# B&R Automation Studio project NAELD004C00R10L518F00 (part 8)

#### Act_OptP0201QueryWorkOrderInfo.st
```iecst
ACTION Act_OptP0201QueryWorkOrderInfo:

	//Mask Magazine Barcode / SlotId
	IF p_tyNtParamCurr.bHermesSvyMagTypeMc = FALSE THEN
		fUIInRtStatOff(ADR(tyP0201OpsTravLifter.tyQueryWorkOrderInfo.tyBitmapMask.uiMaskRtStat)); //show the mask
	ELSE
		fUIInRtStatHide(ADR(tyP0201OpsTravLifter.tyQueryWorkOrderInfo.tyBitmapMask.uiMaskRtStat)); //hide the mask
	END_IF

	//Mask Barcode Scanner
	IF p_tyNtParamCurr.bHermesScannerPrep = TRUE AND p_tyMcParamCurr.bHermesScannerEn = TRUE THEN
		fUIInRtStatHide(ADR(tyP0201OpsTravLifter.tyQueryWorkOrderInfo.tyBtnBarcodeScanner.uiMaskRtStat)); //hide the mask
	ELSE
		fUIInRtStatOff(ADR(tyP0201OpsTravLifter.tyQueryWorkOrderInfo.tyBtnBarcodeScanner.uiMaskRtStat)); //show the mask
	END_IF

	IF 	EDGEPOS (tyP0201OpsTravLifter.tyQueryWorkOrderInfo.tyBtnBarcodeScanner.bValue = TRUE) THEN
		fUIInRtStatHide(ADR(tyP0201OpsTravLifter.tyQueryWorkOrderInfo.tyLyr.uiRtStat)); //hide popup QueryBoardInfo
		fUIInRtStatOff(ADR(tyP0201OpsTravLifter.tyBarcodeScanner.tyLyr.uiRtStat)); //show popup BCScanner
		fUIInRtStatHide(ADR(tyP0201OpsTravLifter.tyBarcodeScanner.tyBtnMagazine.uiMaskRtStat)); //hide Mask Magazine
		fUIInRtStatOff(ADR(tyP0201OpsTravLifter.tyBarcodeScanner.tyBtnTop.uiMaskRtStat)); //Mask Top
	END_IF

	//Convert
	iSlotId := DINT_TO_INT(tyP0201OpsTravLifter.tyQueryWorkOrderInfo.tyNumSlotId.diValue);

	//Press OK, set bQueryWorkOrderInfo
	IF	tyP0201OpsTravLifter.tyQueryWorkOrderInfo.tyBtnOk.bRtCompl = TRUE THEN

		fUIInRtStatHide(ADR(tyP0201OpsTravLifter.tyQueryWorkOrderInfo.tyLyr.uiRtStat)); //close popup

		IF (tyP0201OpsTravLifter.tyQueryWorkOrderInfo.tyStringMagazineId.sValue <> '') OR (iSlotId <> 0)
			OR (tyP0201OpsTravLifter.tyQueryWorkOrderInfo.tyStringBarcode.sValue <> '') THEN
			bQueryWorkOrderInfo := TRUE;
			tyP0201OpsTravLifter.tyCurrWorkOrderInfo.tyBtnQueryWorkOrderInfo.bValue := TRUE;
		ELSE
			bQueryWorkOrderInfo := FALSE;
			tyP0201OpsTravLifter.tyCurrWorkOrderInfo.tyBtnQueryWorkOrderInfo.bValue := FALSE;
		END_IF

		tyP0201OpsTravLifter.tyQueryWorkOrderInfo.tyBtnOk.bValue := FALSE;

		tyP0201OpsTravLifter.tyQueryWorkOrderInfo.tyBtnOk.bRtCompl := FALSE;

	END_IF

	//Press Cancel
	IF	tyP0201OpsTravLifter.tyQueryWorkOrderInfo.tyBtnCancel.bRtCompl = TRUE THEN

		fUIInRtStatHide(ADR(tyP0201OpsTravLifter.tyQueryWorkOrderInfo.tyLyr.uiRtStat)); //hide
		fUIInRtStatOff(ADR(tyP0201OpsTravLifter.tyCurrWorkOrderInfo.tyLyr.uiRtStat)); //hide

		tyP0201OpsTravLifter.tyQueryWorkOrderInfo.tyBtnCancel.bRtCompl := FALSE;
		tyP0201OpsTravLifter.tyQueryWorkOrderInfo.tyBtnCancel.bValue := FALSE;
	END_IF

END_ACTION
```

#### Act_OptP0201UpdtDat.st
```iecst
ACTION Act_OptP0201UpdtDat:

	//Status
	fbMcStatUpdtTm(IN := TRUE);
	IF fbMcStatUpdtTm.Q = TRUE THEN
		fbMcStatUpdtTm(IN := FALSE);

		IF p_bOpsTravLifLDAWPosDiff THEN
			IF p_tyNtParamCurr.bDSWidthChkPrep AND p_tyMcParamCurr.bDSWidthChkEn AND p_tyDI.bDSWidthChkSen=FALSE THEN
				tyP0201OpsTravLifter.tyOps.tyStringMcStat.sValue	:= 'Width Check Sensor Block Downstream';
			ELSIF p_tyNtParamCurr.bLFPrep AND p_tyMcParamCurr.bLFEn AND p_bLFFollowerDSAllow=FALSE THEN
				IF p_tyMcParamCurr.bSectionLeader THEN
					tyP0201OpsTravLifter.tyOps.tyStringMcStat.sValue	:= 'Section Leader: Block Downstream';
				ELSE
					tyP0201OpsTravLifter.tyOps.tyStringMcStat.sValue	:= 'Leader Issue Block Downstream';
				END_IF

			ELSE
				tyP0201OpsTravLifter.tyOps.tyStringMcStat.sValue	:= p_sOpsTravLifLDStepTxt;
			END_IF
		ELSE
			tyP0201OpsTravLifter.tyOps.tyStringMcStat.sValue	:= p_sOpsTravLifLDStepTxt;
		END_IF
	END_IF

	//Mode
	tyP0201OpsTravLifter.tyOps.tyTxtMod.usiValueIdx	:= p_tyProdRcpCurrRcp2.usiMcMod;

	//Width
	IF p_tyNtParamCurr.bAWPrep = TRUE AND p_tyMcParamCurr.bAWDis = FALSE THEN
		tyP0201OpsTravLifter.tyOps.tyNumWidth.diValue	:= p_tyMcParamCurr.diWidthAtHmPosInUM - p_diAWOpenActualPos;
		tyP0201OpsTravLifter.tyOps.tyNumWidth2.diValue	:= p_tyMcParamCurr.diWidthAtHmPosInUM - p_diAWOpenActualPos;
	ELSE
		tyP0201OpsTravLifter.tyOps.tyNumWidth.diValue	:= p_tyProdRcpCurrRcp2.diWidthInUM;
		tyP0201OpsTravLifter.tyOps.tyNumWidth2.diValue	:= p_tyProdRcpCurrRcp2.diWidthInUM2;
	END_IF

	//Product Info
	IF p_tyNtParamCurr.eProjMag <> LDMagQuadruple THEN
		IF p_tyNtParamCurr.bProjAutoRcpPrep AND p_tyMcParamCurr.bHermesSvyEn THEN
			IF p_ausiSvyMagAccOrder[1] = 10 THEN
				tyP0201OpsTravLifter.tyOps.tyNumMinSltRange.diValue		:= p_diLinkAutoRcpMag1MinSlt;
				tyP0201OpsTravLifter.tyOps.tyNumMaxSltRange.diValue		:= p_diLinkAutoRcpMag1MaxSlt;
				tyP0201OpsTravLifter.tyOps.tyNumPitch.diValue			:= p_diLinkAutoRcpMag1Pitch;
				tyP0201OpsTravLifter.tyOps.tyStringProdNm.sValue		:= p_tyAutoRcpMagRcp[1].sWorkOrderId;
			ELSIF p_ausiSvyMagAccOrder[2] = 10 THEN
				tyP0201OpsTravLifter.tyOps.tyNumMinSltRange.diValue		:= p_diLinkAutoRcpMag2MinSlt;
				tyP0201OpsTravLifter.tyOps.tyNumMaxSltRange.diValue		:= p_diLinkAutoRcpMag2MaxSlt;
				tyP0201OpsTravLifter.tyOps.tyNumPitch.diValue			:= p_diLinkAutoRcpMag2Pitch;
				tyP0201OpsTravLifter.tyOps.tyStringProdNm.sValue		:= p_tyAutoRcpMagRcp[2].sWorkOrderId;
			ELSIF p_ausiSvyMagAccOrder[3] = 10 THEN
				tyP0201OpsTravLifter.tyOps.tyNumMinSltRange.diValue		:= p_diLinkAutoRcpMag3MinSlt;
				tyP0201OpsTravLifter.tyOps.tyNumMaxSltRange.diValue		:= p_diLinkAutoRcpMag3MaxSlt;
				tyP0201OpsTravLifter.tyOps.tyNumPitch.diValue			:= p_diLinkAutoRcpMag3Pitch;
				tyP0201OpsTravLifter.tyOps.tyStringProdNm.sValue		:= p_tyAutoRcpMagRcp[3].sWorkOrderId;
			END_IF
		ELSE //standard
			tyP0201OpsTravLifter.tyOps.tyNumMinSltRange.diValue		:= p_tyProdRcpCurrRcp2.diMinSltValue;
			tyP0201OpsTravLifter.tyOps.tyNumMaxSltRange.diValue		:= p_tyProdRcpCurrRcp2.diMaxSltValue;
			tyP0201OpsTravLifter.tyOps.tyNumPitch.diValue			:= p_tyProdRcpCurrRcp2.diPitch;
			tyP0201OpsTravLifter.tyOps.tyStringProdNm.sValue		:= p_tyProdRcpCurrRcp2.sRcpNm;
		END_IF

		tyP0201OpsTravLifter.tyOps.tyBtnToptoBtm.bValue			:= p_tyProdRcpCurrRcp2.bTopToBtm;

		tyP0201OpsTravLifter.tyOps.tyNumPshrOffset.diValue		:= p_tyProdRcpCurrRcp2.diPshrOffset;
		tyP0201OpsTravLifter.tyOps.tyNumMtrPshrExtSpd.diValue	:= p_tyProdRcpCurrRcp2.diMtrPshrExtSpd;
		tyP0201OpsTravLifter.tyOps.tyNumMtrPshrExtTorq.diValue	:= p_tyProdRcpCurrRcp2.diMtrPshrExtTorq;

	ELSE //quadral
		tyP0201OpsTravLifter.tyOps.tyStringProdNm.sValue		:= p_tyProdRcpCurrRcp2.sRcpNm;
		tyP0201OpsTravLifter.tyOps.tyNumMinSltRange.diValue		:= p_tyProdRcpCurrRcp2.diMinSltValue;
		tyP0201OpsTravLifter.tyOps.tyNumMaxSltRange.diValue		:= p_tyProdRcpCurrRcp2.diMaxSltValue;
		tyP0201OpsTravLifter.tyOps.tyBtnToptoBtm.bValue			:= p_tyProdRcpCurrRcp2.bTopToBtm;
		tyP0201OpsTravLifter.tyOps.tyNumPitch.diValue			:= p_tyProdRcpCurrRcp2.diPitch;

		tyP0201OpsTravLifter.tyOps.tyNumMinSltRange.diValue		:= p_tyProdRcpCurrRcp2.diMinSltValue;
		tyP0201OpsTravLifter.tyOps.tyNumMaxSltRange.diValue		:= p_tyProdRcpCurrRcp2.diMaxSltValue;
		tyP0201OpsTravLifter.tyOps.tyNumPitch.diValue			:= p_tyProdRcpCurrRcp2.diPitch;
	END_IF

	//PCB Status
	IF p_bPullConvHvBrd = TRUE THEN
		tyP0201OpsTravLifter.tyOps.tyBitmapPCB.usiValueIdx	:= 1;
	ELSE
		tyP0201OpsTravLifter.tyOps.tyBitmapPCB.usiValueIdx	:= 0;
	END_IF

	//Product Recipe 254
	tyP0201OpsTravLifter.tyOps.tyHotspotShowLRcp.uiRtStat.0 := NOT(tyP0201OpsTravLifter.tyOps.tyStringProdNm.sValue <> '');

	IF tyP0201OpsTravLifter.tyOps.tyHotspotShowLRcp.bRtCompl = TRUE THEN
		tyP0201OpsTravLifter.tyOps.tyHotspotShowLRcp.bRtCompl := FALSE;

		fUIInRtStatOff(ADR(tyP0201OpsTravLifter.tyRcpPopUp.tyLyr.uiRtStat));

		tyP0201OpsTravLifter.tyRcpPopUp.tyStringInfo.sValue  := p_tyProdRcpCurrRcp1.sRcpNm;

	ELSIF tyP0201OpsTravLifter.tyRcpPopUp.tyHotspotClose.bRtCompl = TRUE THEN
		tyP0201OpsTravLifter.tyRcpPopUp.tyHotspotClose.bRtCompl := FALSE;

		fUIInRtStatHide(ADR(tyP0201OpsTravLifter.tyRcpPopUp.tyLyr.uiRtStat));

	END_IF

END_ACTION
```

#### Act_EntP0202Disp.st
```iecst
ACTION Act_EntP0202Disp:

	//Access Address
	p_tyC0004Navi ACCESS ADR(tyP0202OpsMag1.tyNaviBack);

	p_tyC0005Main ACCESS ADR(tyCommon.tyMain);

	p_tyC0007Notif ACCESS ADR(tyCommon.tyNotif);

	p_tyC0008MsgBox ACCESS ADR(tyP0202OpsMag1.tyMsgBoxHide);

	p_tyC0009Info ACCESS ADR(tyCommon.tyInfo);

	p_tyC0011RcpPopUp ACCESS ADR(tyP0202OpsMag1.tyRcpPopUp);

	p_tyP0202Ops ACCESS ADR(tyP0202OpsMag1.tyOps);
	p_tyP0202IOMonitor ACCESS ADR(tyP0202OpsMag1.tyIOMonitor);
	p_tyP0202BypsInitConv ACCESS ADR(tyP0202OpsMag1.tyBypsInitConv);
	p_tyP0202Param ACCESS ADR(tyP0202OpsMag1.tyParam);

	//Display
	fUIInRtStatHide(ADR(tyP0202OpsMag1.tyIOMonitor.tyLyr.uiRtStat));
	fUIInRtStatHide(ADR(tyP0202OpsMag1.tyParam.tyLyr.uiRtStat));

	tyP0202OpsMag1.tyOps.tyBtnChgParam.uiRtStat.0	:= NOT(p_tyMcParamCurr.bChgParamEn);
	tyP0202OpsMag1.tyParam.tyNumMaxSlt.diValueMax	:= p_tyMagRcpCurrRcp.diTtlSlt;

	IF p_tyNtParamCurr.bMagAutoVerifyPrep = FALSE THEN
		tyP0202OpsMag1.tyIOMonitor.tyBtnMag1FixedClmpRS.usiTxtIdx	:= 75;
		tyP0202OpsMag1.tyIOMonitor.tyBtnMag1FixedUnclmpRS.usiTxtIdx:= 75;
		tyP0202OpsMag1.tyIOMonitor.tyBtnMag1RmtClmpRS.usiTxtIdx	:= 0;
		tyP0202OpsMag1.tyIOMonitor.tyBtnMag1RmtUnclmpRS.usiTxtIdx:= 0;
		tyP0202OpsMag1.tyIOMonitor.tyBtnMag1FixedClampCtrl.usiTxtIdx:= 41;
		tyP0202OpsMag1.tyIOMonitor.tyBtnMag1RemoteClampCtrl.usiTxtIdx:= 18;
	ELSE
		tyP0202OpsMag1.tyIOMonitor.tyBtnMag1FixedClmpRS.usiTxtIdx	:= 75;
		tyP0202OpsMag1.tyIOMonitor.tyBtnMag1FixedUnclmpRS.usiTxtIdx:= 75;
		tyP0202OpsMag1.tyIOMonitor.tyBtnMag1RmtClmpRS.usiTxtIdx	:= 0;
		tyP0202OpsMag1.tyIOMonitor.tyBtnMag1RmtUnclmpRS.usiTxtIdx:= 0;
		tyP0202OpsMag1.tyIOMonitor.tyBtnMag1FixedClampCtrl.usiTxtIdx:= 41;
		tyP0202OpsMag1.tyIOMonitor.tyBtnMag1RemoteClampCtrl.usiTxtIdx:= 18;

	END_IF

	fUIInRtStatHide(ADR(tyP0202OpsMag1.tyOps.tyBtnAIVWifi.uiRtStat));
	fUIInRtStatHide(ADR(tyP0202OpsMag1.tyOps.tyTxtLblAIV.uiRtStat));

	tyP0202OpsMag1.tyParam.tyNumMaxSlt.diValueMax	:= p_tyMagRcpCurrRcp.diTtlSlt;

END_ACTION
```

#### Act_OptP0202UpdtDat.st
```iecst
ACTION Act_OptP0202UpdtDat:

	//Status
	fbMcStatUpdtTm(IN := TRUE);
	IF fbMcStatUpdtTm.Q = TRUE THEN
		fbMcStatUpdtTm(IN := FALSE);

		IF p_tyNtParamCurr.bProjLifterMagPlatform THEN
			tyP0202OpsMag1.tyOps.tyStringMcStat.sValue	:= p_sOpsLifMagLDStepTxt;
		ELSE
			tyP0202OpsMag1.tyOps.tyStringMcStat.sValue	:= p_sOpsMagConvLD1StepTxt;
		END_IF

	END_IF

	//Mode
	tyP0202OpsMag1.tyOps.tyTxtMod.usiValueIdx	:= p_tyProdRcpCurrRcp1.usiMcMod;

	//Width
	IF p_tyNtParamCurr.bAWPrep = TRUE AND p_tyMcParamCurr.bAWDis = FALSE THEN
		tyP0202OpsMag1.tyOps.tyNumWidth.diValue	:= p_tyMcParamCurr.diWidthAtHmPosInUM - p_diAWOpenActualPos;
		tyP0202OpsMag1.tyOps.tyNumWidth2.diValue	:= p_tyMcParamCurr.diWidthAtHmPosInUM - p_diAWOpenActualPos;
	ELSE
		tyP0202OpsMag1.tyOps.tyNumWidth.diValue	:= p_tyProdRcpCurrRcp1.diWidthInUM;
		tyP0202OpsMag1.tyOps.tyNumWidth2.diValue	:= p_tyProdRcpCurrRcp1.diWidthInUM2;
	END_IF

	//Program Info
	IF p_tyNtParamCurr.eProjMag <> LDMagQuadruple THEN
		IF p_tyNtParamCurr.bProjAutoRcpPrep AND p_tyMcParamCurr.bHermesSvyEn THEN
			tyP0202OpsMag1.tyOps.tyNumMinSltRange.diValue		:= p_diLinkAutoRcpMag1MinSlt;
			tyP0202OpsMag1.tyOps.tyNumMaxSltRange.diValue		:= p_diLinkAutoRcpMag1MaxSlt;
			tyP0202OpsMag1.tyOps.tyNumPitch.diValue				:= p_diLinkAutoRcpMag1Pitch;
			tyP0202OpsMag1.tyOps.tyStringProdNm.sValue			:= p_tyAutoRcpMagRcp[1].sWorkOrderId;
		ELSE
			tyP0202OpsMag1.tyOps.tyNumMinSltRange.diValue		:= p_tyProdRcpCurrRcp2.diMinSltValue;
			tyP0202OpsMag1.tyOps.tyNumMaxSltRange.diValue		:= p_tyProdRcpCurrRcp2.diMaxSltValue;
			tyP0202OpsMag1.tyOps.tyNumPitch.diValue				:= p_tyProdRcpCurrRcp2.diPitch;
			tyP0202OpsMag1.tyOps.tyStringProdNm.sValue		:= p_tyProdRcpCurrRcp2.sRcpNm;
		END_IF
		tyP0202OpsMag1.tyOps.tyBtnToptoBtm.bValue			:= p_tyProdRcpCurrRcp2.bTopToBtm;
		//Magazine Info
		tyP0202OpsMag1.tyOps.tyStringMagNm.sValue	:= p_tyMagRcpCurrRcp.sRcpNm;
	ELSE
		CASE p_tyProdRcpCurrRcp2.usiMcMod OF
			0,2:
				tyP0202OpsMag1.tyOps.tyStringProdNm.sValue		:= p_tyProdRcpCurrRcp2.sRcpNm;
				tyP0202OpsMag1.tyOps.tyNumMinSltRange.diValue		:= p_tyProdRcpCurrRcp2.diMinSltValue;
				tyP0202OpsMag1.tyOps.tyNumMaxSltRange.diValue		:= p_tyProdRcpCurrRcp2.diMaxSltValue;
				tyP0202OpsMag1.tyOps.tyBtnToptoBtm.bValue			:= p_tyProdRcpCurrRcp2.bTopToBtm;
				tyP0202OpsMag1.tyOps.tyNumPitch.diValue			:= p_tyProdRcpCurrRcp2.diPitch;
				//Magazine Info
				tyP0202OpsMag1.tyOps.tyStringMagNm.sValue	:= p_tyMagRcpCurrRcp.sRcpNm;
			1:

				tyP0202OpsMag1.tyOps.tyStringProdNm.sValue		:= p_tyProdRcpCurrRcp2.sRcpNm;
				tyP0202OpsMag1.tyOps.tyNumMinSltRange.diValue		:= p_tyProdRcpCurrRcp2.diMinSltValueRear;
				tyP0202OpsMag1.tyOps.tyNumMaxSltRange.diValue		:= p_tyProdRcpCurrRcp2.diMaxSltValueRear;
				tyP0202OpsMag1.tyOps.tyBtnToptoBtm.bValue			:= p_tyProdRcpCurrRcp2.bTopToBtm;
				tyP0202OpsMag1.tyOps.tyNumPitch.diValue			:= p_tyProdRcpCurrRcp2.diPitchRear;
				//Magazine Info
				tyP0202OpsMag1.tyOps.tyStringMagNm.sValue	:= p_tyMagRcpCurrRcp1.sRcpNm;
		END_CASE
	END_IF
	//Magazine Info
//	tyP0202OpsMag1.tyOps.tyStringMagNm.sValue	:= p_tyMagRcpCurrRcp.sRcpNm;

	IF p_bBuffer1MagPresent = TRUE THEN
		tyP0202OpsMag1.tyOps.tyNumMag1AvlQty.diValue	:= p_tyBuffer1BffrStat.diTtlGdBrd + p_tyBuffer1BffrStat.diTtlBadBrd;
		tyP0202OpsMag1.tyOps.tyNumMag1TtlSlt.diValue	:= p_tyBuffer1BffrStat.diTtlBrdCap;
	ELSE
		tyP0202OpsMag1.tyOps.tyNumMag1AvlQty.diValue	:= 0;
		tyP0202OpsMag1.tyOps.tyNumMag1TtlSlt.diValue	:= 0;
	END_IF

	//Magazine Present States
	IF p_bBuffer1MagPresent = TRUE THEN

		IF p_tyBuffer1BffrStat.bBffrFull = TRUE THEN
			tyP0202OpsMag1.tyOps.tyTxtMag1Stat.usiValueIdx := 2;
			tyP0202OpsMag1.tyOps.tyTxtMag1Stat.usiColor	   := 0;
		ELSIF p_tyBuffer1BffrStat.bBffrMty = TRUE THEN
			tyP0202OpsMag1.tyOps.tyTxtMag1Stat.usiValueIdx := 1;
			tyP0202OpsMag1.tyOps.tyTxtMag1Stat.usiColor	   := 1;
		ELSE
			tyP0202OpsMag1.tyOps.tyTxtMag1Stat.usiValueIdx := 3;
			tyP0202OpsMag1.tyOps.tyTxtMag1Stat.usiColor	   := 0;
		END_IF

	ELSE
		tyP0202OpsMag1.tyOps.tyTxtMag1Stat.usiValueIdx := 0;
		tyP0202OpsMag1.tyOps.tyTxtMag1Stat.usiColor	   := 1;
	END_IF

	//Product Recipe 254
	tyP0202OpsMag1.tyOps.tyHotspotShowLRcp.uiRtStat.0 := NOT(tyP0202OpsMag1.tyOps.tyStringProdNm.sValue <> '');

	IF tyP0202OpsMag1.tyOps.tyHotspotShowLRcp.bRtCompl = TRUE THEN
		tyP0202OpsMag1.tyOps.tyHotspotShowLRcp.bRtCompl := FALSE;

		fUIInRtStatOff(ADR(tyP0202OpsMag1.tyRcpPopUp.tyLyr.uiRtStat));

		tyP0202OpsMag1.tyRcpPopUp.tyStringInfo.sValue  := p_tyProdRcpCurrRcp1.sRcpNm;

	ELSIF tyP0202OpsMag1.tyRcpPopUp.tyHotspotClose.bRtCompl = TRUE THEN
		tyP0202OpsMag1.tyRcpPopUp.tyHotspotClose.bRtCompl := FALSE;

		fUIInRtStatHide(ADR(tyP0202OpsMag1.tyRcpPopUp.tyLyr.uiRtStat));

	END_IF

END_ACTION
```

#### Act_OptP0202IOMonitor.st
```iecst
ACTION Act_OptP0202IOMonitor:

	IF tyP0202OpsMag1.tyOps.tyHotspotIOMonitor.bRtCompl = TRUE THEN
		tyP0202OpsMag1.tyOps.tyHotspotIOMonitor.bRtCompl	:= FALSE;

		fUIInRtStatOff(ADR(tyP0202OpsMag1.tyIOMonitor.tyLyr.uiRtStat));

		p_tyC0004Navi ACCESS ADR(tyP0202OpsMag1.tyNaviHide);

	ELSIF tyP0202OpsMag1.tyIOMonitor.tyHotspotClose.bRtCompl = TRUE THEN
		tyP0202OpsMag1.tyIOMonitor.tyHotspotClose.bRtCompl	:= FALSE;

		fUIInRtStatHide(ADR(tyP0202OpsMag1.tyIOMonitor.tyLyr.uiRtStat));

		p_tyC0004Navi ACCESS ADR(tyP0202OpsMag1.tyNaviBack);

	END_IF

	IF tyP0202OpsMag1.tyIOMonitor.tyLyr.uiRtStat.0 = FALSE THEN

		//Digital Input
		tyP0202OpsMag1.tyIOMonitor.tyBtnSafetyRlySig.bValue				:= p_tyDI.bSafetyRlySig;
		tyP0202OpsMag1.tyIOMonitor.tyBtnEStop.bValue					:= p_tyDI.bEStopSig;
		tyP0202OpsMag1.tyIOMonitor.tyBtnCoverSWSig.bValue				:= p_tyDI.bCoverSWSig;
		tyP0202OpsMag1.tyIOMonitor.tyBtnDSBA.bValue						:= p_tyDI.bDSBA;
		tyP0202OpsMag1.tyIOMonitor.tyBtnDSBB.bValue						:= p_tyDI.bDSBB;
		tyP0202OpsMag1.tyIOMonitor.tyBtnMag1FixedClmpRS.bValue			:= p_tyDI.bMag1FixedClampRS;
		tyP0202OpsMag1.tyIOMonitor.tyBtnMag1FixedUnclmpRS.bValue		:= p_tyDI.bMag1FixedUnclampRS;
		tyP0202OpsMag1.tyIOMonitor.tyBtnMag1RmtClmpRS.bValue			:= p_tyDI.bMag1RemoteClampRS;
		tyP0202OpsMag1.tyIOMonitor.tyBtnMag1RmtUnclmpRS.bValue			:= p_tyDI.bMag1RemoteUnclampRS;
		tyP0202OpsMag1.tyIOMonitor.tyBtnMag1ConvEntrySen.bValue			:= p_tyDI.bMagConvEntSen1;
		tyP0202OpsMag1.tyIOMonitor.tyBtnMag1PresentSen.bValue			:= p_tyDI.bMagPresentSen1;
		tyP0202OpsMag1.tyIOMonitor.tyBtnMag1AIVInPosSen1.bValue			:= p_tyDI.bMag1AGVInPosSen1;
		tyP0202OpsMag1.tyIOMonitor.tyBtnMag1AIVInPosSen2.bValue			:= p_tyDI.bMag1AGVInPosSen2;
		tyP0202OpsMag1.tyIOMonitor.tyBtnMag1OrientationChkSen1.bValue	:= p_tyDI.bMag1OrientChkSen1;
		tyP0202OpsMag1.tyIOMonitor.tyBtnMag1OrientationChkSen2.bValue	:= p_tyDI.bMag1OrientChkSen2;

		tyP0202OpsMag1.tyIOMonitor.tyBtnSelUnclampRS.bValue				:= p_tyDI.bMag1SelUnClampRS;

		tyP0202OpsMag1.tyIOMonitor.tyBtnCAB717Sen.bValue				:= p_tyDI.bMagConvCAB717MagSen1;
		tyP0202OpsMag1.tyIOMonitor.tyBtnHeightSen.bValue				:= p_tyDI.bMagConvHeightSen1 OR p_tyDI.bHighMagDetSen1;
		tyP0202OpsMag1.tyIOMonitor.tyBtnMagSmallSen.bValue				:= p_tyDI.bMagConvSmallMagSen1;
		tyP0202OpsMag1.tyIOMonitor.tyBtnMagLargeSen.bValue				:= p_tyDI.bMagConvLargeMagSen1;
		tyP0202OpsMag1.tyIOMonitor.tyBtnMagDetSen.bValue				:= p_tyDI.bMag1FixedSideDetect;
		tyP0202OpsMag1.tyIOMonitor.tyBtnTrllyExtRS.bValue				:= p_tyDI.bTrolleyExtRS1;
		tyP0202OpsMag1.tyIOMonitor.tyBtnTrllyPresentSen.bValue			:= p_tyDI.bTrolleyPreSen1;
		tyP0202OpsMag1.tyIOMonitor.tyBtnSltLckSen.bValue				:= p_tyDI.bSlotLckSenMag1;

		//Digital Output
		tyP0202OpsMag1.tyIOMonitor.tyBtnSafetyRlyRst.bValue				:= p_tyDO.bSafetyRlyRst;
		tyP0202OpsMag1.tyIOMonitor.tyBtnTLGreen.bValue					:= p_tyDO.bTLGreen;
		tyP0202OpsMag1.tyIOMonitor.tyBtnTLAmber.bValue					:= p_tyDO.bTLAmber;
		tyP0202OpsMag1.tyIOMonitor.tyBtnTLRed.bValue					:= p_tyDO.bTLRed;
		tyP0202OpsMag1.tyIOMonitor.tyBtnBuzzer.bValue					:= p_tyDO.bBuzzer;
		tyP0202OpsMag1.tyIOMonitor.tyBtnDBAA.bValue						:= p_tyDO.bDBAA;
		tyP0202OpsMag1.tyIOMonitor.tyBtnDBAB.bValue						:= p_tyDO.bDBAB;
		tyP0202OpsMag1.tyIOMonitor.tyBtnMag1FixedClampCtrl.bValue		:= p_tyDO.bMag1FixedClampCtrl;
		tyP0202OpsMag1.tyIOMonitor.tyBtnMag1RemoteClampCtrl.bValue		:= p_tyDO.bMag1RemoteClampCtrl;
		tyP0202OpsMag1.tyIOMonitor.tyBtnMag1ConvMtrIn.bValue			:= p_tyDO.bMag1ConvMtrIn;
		tyP0202OpsMag1.tyIOMonitor.tyBtnMag1ConvMtrOut.bValue			:= p_tyDO.bMag1ConvMtrOut;
		tyP0202OpsMag1.tyIOMonitor.tyBtnMagSelClampCtrl.bValue			:= p_tyDO.bMag1SelClampCtrl;
		tyP0202OpsMag1.tyIOMonitor.tyBtnTrllyExtCtrl.bValue				:= p_tyDO.bTrolleyLckCtrl1;
	END_IF

END_ACTION
```

#### Act_OptP0202AIVDat.st
```iecst
ACTION Act_OptP0202AIVDat:

	//Show Change Mag Button only in Manual Exchane Mode
	tyP0202OpsMag1.tyOps.tyBtnChgMag.uiRtStat.0 := p_tyMcParamCurr.eMagExMode = McSetMagXcAutoMode AND p_tyMcParamCurr.eAGVComProtocol <> McSetAGVCommDisabled  OR p_tyNtParamCurr.bProjLifterMagPlatform;;
	tyP0202OpsMag1.tyOps.tyBitmapChgMag.uiRtStat.0 := p_tyMcParamCurr.eMagExMode = McSetMagXcAutoMode AND p_tyMcParamCurr.eAGVComProtocol <> McSetAGVCommDisabled  OR p_tyNtParamCurr.bProjLifterMagPlatform;;
	//LED Wifi
	tyP0202OpsMag1.tyOps.tyBtnAIVWifi.bValue	:= p_bAGVOnline;

	//Change Magazine
	IF p_tyNtParamCurr.bProjBtnInsertRmvMag = TRUE THEN

		IF EDGENEG(p_bOpsStatusRun) THEN
			bNewMag1	:= FALSE;
			tyP0202OpsMag1.tyOps.tyBtnChgMag.bRtLk	:= FALSE;
			tyP0202OpsMag1.tyOps.tyBtnChgMag.bRtCompl	:= FALSE;
			tyP0202OpsMag1.tyOps.tyBtnChgMag.bValue		:= FALSE;
		END_IF

		IF tyP0202OpsMag1.tyOps.tyBtnChgMag.bRtCompl = TRUE THEN
			tyP0202OpsMag1.tyOps.tyBitmapChgMag.usiValueIdx	:= 1;
			tyP0202OpsMag1.tyOps.tyBtnChgMag.bRtLk := TRUE;
			IF 	p_bOpsMagConvLD1NewMagAllw OR p_bOpsMagConvLD1RlsMagAllw OR p_bOpsMagConvLD1RlsMagUmask THEN
				tyP0202OpsMag1.tyOps.tyBtnChgMag.bRtCompl	:= FALSE;
				bNewMag1	:= p_bOpsMagConvLD1NewMagAllw;
				bRlsMag1	:= p_bOpsMagConvLD1RlsMagAllw;
				bEjectMag1  := p_bOpsMagConvLD1ExtMes;
			END_IF
		END_IF

		IF bNewMag1 = TRUE THEN
			tyP0202OpsMag1.tyOps.tyBitmapChgMag.usiValueIdx	:= 1;

			IF p_tyDI.bMag1FixedUnclampRS = FALSE OR p_eMagConv2Clp1Status = Error THEN
				bNewMag1	:= FALSE;
				tyP0202OpsMag1.tyOps.tyBtnChgMag.bValue	:= FALSE;
				tyP0202OpsMag1.tyOps.tyBtnChgMag.bRtLk	:= FALSE;
				tyP0202OpsMag1.tyOps.tyBitmapChgMag.usiValueIdx	:= 0;
			END_IF

		ELSIF bRlsMag1 = TRUE OR bEjectMag1 THEN
				tyP0202OpsMag1.tyOps.tyBitmapChgMag.usiValueIdx	:= 1;
			IF p_tyNtParamCurr.eCustomerReq = Siemens OR p_tyNtParamCurr.eCustomerReq = We_Fabricate THEN
				IF p_bOpsMagConvLD1RlsMagUmask THEN // siemens , read -1 or write TO
					IF p_tyNtParamCurr.eCustomerReq = We_Fabricate THEN
						//bRlsMag1	:= FALSE;
						tyP0202OpsMag1.tyOps.tyBitmapChgMag.usiValueIdx	:= 0;
					END_IF
					tyP0202OpsMag1.tyOps.tyBtnChgMag.bValue	:= FALSE;
					tyP0202OpsMag1.tyOps.tyBtnChgMag.bRtLk	:= FALSE;
				ELSIF p_bOpsMagConvLD1ExtMes THEN //2nd press to eject mag
					bEjectMag1	:= FALSE;
					bRlsMag1	:= FALSE;
					tyP0202OpsMag1.tyOps.tyBtnChgMag.bValue	:= FALSE;
					tyP0202OpsMag1.tyOps.tyBtnChgMag.bRtLk	:= FALSE;
					tyP0202OpsMag1.tyOps.tyBitmapChgMag.usiValueIdx	:= 0;
				ELSIF (p_tyDI.bMag1FixedUnclampRS = TRUE AND p_tyDI.bMagPresentSen1 = FALSE) AND p_tyMcParamCurr.eDSCommA = 0 THEN//smema
					bRlsMag1	:= FALSE;
					tyP0202OpsMag1.tyOps.tyBtnChgMag.bValue	:= FALSE;
					tyP0202OpsMag1.tyOps.tyBtnChgMag.bRtLk	:= FALSE;
					tyP0202OpsMag1.tyOps.tyBitmapChgMag.usiValueIdx	:= 0;
				END_IF

			ELSIF (p_tyDI.bMag1FixedUnclampRS = TRUE AND p_tyDI.bMagPresentSen1 = FALSE)THEN
				bRlsMag1	:= FALSE;
				tyP0202OpsMag1.tyOps.tyBtnChgMag.bValue	:= FALSE;
				tyP0202OpsMag1.tyOps.tyBtnChgMag.bRtLk	:= FALSE;
				tyP0202OpsMag1.tyOps.tyBitmapChgMag.usiValueIdx	:= 0;
			END_IF

		END_IF

		IF p_tyDI.bMagPresentSen1 AND p_tyDI.bMagConvEntSen1 = FALSE THEN
			tyP0202OpsMag1.tyOps.tyBtnChgMag.usiTxtIdx	:= 1;
		ELSE
			tyP0202OpsMag1.tyOps.tyBtnChgMag.usiTxtIdx	:= 0;
			tyP0202OpsMag1.tyOps.tyBtnChgMag.uiMaskRtStat := TRUE;
			IF EDGEPOS(tyP0202OpsMag1.tyOps.tyBtnChgMag.usiTxtIdx =0) THEN
				tyP0202OpsMag1.tyOps.tyBitmapChgMag.usiValueIdx	:= 0;
			END_IF
		END_IF

//		tyP0202OpsMag1.tyOps.tyBtnChgMag.uiMaskRtStat.0	:= p_bOpsMagConvLD1NewMagAllw OR p_bOpsMagConvLD1RlsMagAllw OR p_bOpsMagConvLD1RlsMagUmask;// OR p_tyDI.bInShutterCloseRS;
	END_IF

END_ACTION
```

#### Act_OptP0202ChgParam.st
```iecst
ACTION Act_OptP0202ChgParam:

	tyP0202OpsMag1.tyParam.tyNumMinSlt.diValueMax		:= tyP0202OpsMag1.tyParam.tyNumMaxSlt.diValue;
	tyP0202OpsMag1.tyParam.tyNumMaxSlt.diValueMin		:= tyP0202OpsMag1.tyParam.tyNumMinSlt.diValue;
	tyP0202OpsMag1.tyParam.tyNumPitch.diValueMax		:= tyP0202OpsMag1.tyParam.tyNumMaxSlt.diValue - tyP0202OpsMag1.tyParam.tyNumMinSlt.diValue + 1;
	tyP0202OpsMag1.tyParam.tyNumPitch.diValueMin		:= 1;

	tyP0202OpsMag1.tyParam.tyNumMinSltRear.diValueMax		:= tyP0202OpsMag1.tyParam.tyNumMaxSltRear.diValue;
	tyP0202OpsMag1.tyParam.tyNumMaxSltRear.diValueMin		:= tyP0202OpsMag1.tyParam.tyNumMinSltRear.diValue;
	tyP0202OpsMag1.tyParam.tyNumPitchRear.diValueMax		:= tyP0202OpsMag1.tyParam.tyNumMaxSltRear.diValue - tyP0202OpsMag1.tyParam.tyNumMinSltRear.diValue + 1;
	tyP0202OpsMag1.tyParam.tyNumPitchRear.diValueMin		:= 1;

	tyP0202OpsMag1.tyParam.tyNumMtrPshrExtSpd.diValueMin	:= p_tyNtParamCurr.tyProdRcpMtrPshrExtSpd.diMin;
	tyP0202OpsMag1.tyParam.tyNumMtrPshrExtSpd.diValueMax	:= p_tyNtParamCurr.tyProdRcpMtrPshrExtSpd.diMax;
	tyP0202OpsMag1.tyParam.tyNumMtrPshrExtTorq.diValueMin	:= p_tyNtParamCurr.tyProdRcpMtrPshrExtTorq.diMin;
	tyP0202OpsMag1.tyParam.tyNumMtrPshrExtTorq.diValueMax	:= p_tyNtParamCurr.tyProdRcpMtrPshrExtTorq.diMax;
	tyP0202OpsMag1.tyParam.tyNumPshrOffset.diValueMin		:= -(p_tyProdRcpCurrRcp2.diWidthInUM/2-p_tyMcParamCurr.diAWPusherAtHmPosInUM-5000 );
	tyP0202OpsMag1.tyParam.tyNumPshrOffset.diValueMax		:= (p_tyProdRcpCurrRcp2.diWidthInUM/2-p_tyMcParamCurr.diAWPusherAtHmPosInUM-5000 );

	//Control
	IF tyP0202OpsMag1.tyOps.tyBtnChgParam.bRtCompl = TRUE THEN
		tyP0202OpsMag1.tyOps.tyBtnChgParam.bRtCompl	:= FALSE;

		tyProdRcpCurrRcpWr	:= p_tyProdRcpCurrRcp0;

		tyP0202OpsMag1.tyParam.tyDrpDnMcMode.usiValueIdx	:= p_tyProdRcpCurrRcp0.usiMcMod;
		tyP0202OpsMag1.tyParam.tyNumMinSlt.diValue	:= p_tyProdRcpCurrRcp0.diMinSltValue;
		tyP0202OpsMag1.tyParam.tyNumMaxSlt.diValue	:= p_tyProdRcpCurrRcp0.diMaxSltValue;
		tyP0202OpsMag1.tyParam.tyNumPitch.diValue		:= p_tyProdRcpCurrRcp0.diPitch;

		tyP0202OpsMag1.tyParam.tyNumMinSltRear.diValue	:= p_tyProdRcpCurrRcp0.diMinSltValueRear;
		tyP0202OpsMag1.tyParam.tyNumMaxSltRear.diValue	:= p_tyProdRcpCurrRcp0.diMaxSltValueRear;
		tyP0202OpsMag1.tyParam.tyNumPitchRear.diValue		:= p_tyProdRcpCurrRcp0.diPitchRear;

		tyP0202OpsMag1.tyParam.tyNumMtrPshrExtSpd.diValue		:= p_tyProdRcpCurrRcp0.diMtrPshrExtSpd;
		tyP0202OpsMag1.tyParam.tyNumMtrPshrExtTorq.diValue	:= p_tyProdRcpCurrRcp0.diMtrPshrExtTorq;
		tyP0202OpsMag1.tyParam.tyNumPshrOffset.diValue		:= p_tyProdRcpCurrRcp0.diPshrOffset;

		fUIInRtStatOff(ADR(tyP0202OpsMag1.tyParam.tyLyr.uiRtStat));

	END_IF

	tyP0202OpsMag1.tyOps.tyBtnChgParam.bValue		:= tyP0202OpsMag1.tyParam.tyLyr.uiRtStat.0 = FALSE;

	IF tyP0202OpsMag1.tyParam.tyLyr.uiRtStat.0 = FALSE THEN

		IF tyP0202OpsMag1.tyParam.tyBtnSave.bRtCompl = TRUE THEN

			tyProdRcpCurrRcpWr.usiMcMod	:= tyP0202OpsMag1.tyParam.tyDrpDnMcMode.usiValueIdx;
			tyProdRcpCurrRcpWr.diMinSltValue := tyP0202OpsMag1.tyParam.tyNumMinSlt.diValue;
			tyProdRcpCurrRcpWr.diMaxSltValue := tyP0202OpsMag1.tyParam.tyNumMaxSlt.diValue;
			tyProdRcpCurrRcpWr.diPitch := tyP0202OpsMag1.tyParam.tyNumPitch.diValue;

			tyProdRcpCurrRcpWr.diMinSltValueRear := tyP0202OpsMag1.tyParam.tyNumMinSltRear.diValue;
			tyProdRcpCurrRcpWr.diMaxSltValueRear := tyP0202OpsMag1.tyParam.tyNumMaxSltRear.diValue;
			tyProdRcpCurrRcpWr.diPitchRear := tyP0202OpsMag1.tyParam.tyNumPitchRear.diValue;

			tyProdRcpCurrRcpWr.diMtrPshrExtSpd := tyP0202OpsMag1.tyParam.tyNumMtrPshrExtSpd.diValue;
			tyProdRcpCurrRcpWr.diMtrPshrExtTorq := tyP0202OpsMag1.tyParam.tyNumMtrPshrExtTorq.diValue;
			tyProdRcpCurrRcpWr.diPshrOffset := tyP0202OpsMag1.tyParam.tyNumPshrOffset.diValue;

			eProdRcpAct	:= ProdRcpActWriteCurrRcpParam;

			IF p_eProdRcpStatus = Done AND p_eProdRcpStat = ProdRcpActWriteCurrRcpParam THEN
				eProdRcpAct	:= ProdRcpActIdle;

				//UIP0400
				tyP0400ProdSel.tyProdSel.tyTxtMcMode.usiValueIdx	:= p_tyProdRcpCurrRcp0.usiMcMod;

				tyP0400ProdSel.tyProdSel.tyNumMinSlt.diValue	:= p_tyProdRcpCurrRcp0.diMinSltValue;
				tyP0400ProdSel.tyProdSel.tyNumMaxSlt.diValue	:= p_tyProdRcpCurrRcp0.diMaxSltValue;
				tyP0400ProdSel.tyProdSel.tyNumPitch.diValue		:= p_tyProdRcpCurrRcp0.diPitch;

				tyP0400ProdSel.tyProdSel.tyNumMinSltRear.diValue	:= p_tyProdRcpCurrRcp0.diMinSltValueRear;
				tyP0400ProdSel.tyProdSel.tyNumMaxSltRear.diValue	:= p_tyProdRcpCurrRcp0.diMaxSltValueRear;
				tyP0400ProdSel.tyProdSel.tyNumPitchRear.diValue		:= p_tyProdRcpCurrRcp0.diPitchRear;

				tyP0400ProdSel.tyProdSel.tyNumMtrPshrExtSpd.diValue		:= p_tyProdRcpCurrRcp0.diMtrPshrExtSpd;
				tyP0400ProdSel.tyProdSel.tyNumMtrPshrExtTorq.diValue	:= p_tyProdRcpCurrRcp0.diMtrPshrExtTorq;
				tyP0400ProdSel.tyProdSel.tyNumPshrOffset.diValue		:= p_tyProdRcpCurrRcp0.diPshrOffset;

				tyP0202OpsMag1.tyParam.tyBtnSave.bRtCompl			:= FALSE;
				tyP0202OpsMag1.tyParam.tyBtnSave.bValue				:= FALSE;

				fUIInRtStatHide(ADR(tyP0202OpsMag1.tyParam.tyLyr.uiRtStat));

			ELSIF p_eProdRcpStatus = Error THEN
				p_tyC0008MsgBox ACCESS ADR(tyP0202OpsMag1.tyMsgBoxSaveErr);

				IF tyP0202OpsMag1.tyMsgBoxSaveErr.tyBtnNo.bRtCompl = TRUE THEN
					tyP0202OpsMag1.tyMsgBoxSaveErr.tyBtnNo.bRtCompl	:= FALSE;
					tyP0202OpsMag1.tyMsgBoxSaveErr.tyBtnNo.bValue	:= FALSE;

					p_tyC0008MsgBox ACCESS ADR(tyP0202OpsMag1.tyMsgBoxHide);

					//Restore Param
					tyProdRcpCurrRcpWr	:= p_tyProdRcpCurrRcp2;

					tyP0202OpsMag1.tyParam.tyBtnSave.bRtCompl		:= FALSE;
					tyP0202OpsMag1.tyParam.tyBtnSave.bValue			:= FALSE;

					fUIInRtStatHide(ADR(tyP0202OpsMag1.tyParam.tyLyr.uiRtStat));

				END_IF

			END_IF

		ELSIF tyP0202OpsMag1.tyParam.tyBtnCancel.bRtCompl = TRUE THEN
			tyP0202OpsMag1.tyParam.tyBtnCancel.bRtCompl				:= FALSE;
			tyP0202OpsMag1.tyParam.tyBtnCancel.bValue				:= FALSE;

			fUIInRtStatHide(ADR(tyP0202OpsMag1.tyParam.tyLyr.uiRtStat));

		END_IF

	END_IF

	//Mask
	tyP0202OpsMag1.tyOps.tyBtnChgParam.uiMaskRtStat.0	:= p_tyUsrMgmtCurrAccessRgt.bChgParam AND p_bOpsStatusStop;

END_ACTION
```

#### Act_OptP0202InsertRmvMag.st
```iecst
ACTION Act_OptP0202InsertRmvMag:

	//Insert & Removed Magazine Manually Without Button Control
//	IF p_tyNtParamCurr.bProjBtnInsertRmvMag = FALSE THEN
//
//		IF p_bOpsStatusRun AND p_bOpsMagConvLD1InitDone THEN
//
//			fbMag1EntrySenOnTm(IN := p_tyDI.bMagPresentSen1 OR p_tyDI.bMagConvEntSen1);
//
//			IF bNewMag1 = FALSE AND bRlsMag1 = FALSE THEN
//				IF p_bOpsMagConvLD1NewMagAllw AND fbMag1EntrySenOnTm.Q AND NOT p_bOpsMagConvLD1MagExitedWait THEN
//					bNewMag1	:= TRUE;
//				END_IF
//
//				IF p_bOpsMagConvLD1RlsMagAllw AND p_tyDI.bMagPresentSen1 AND p_tyDI.bInShutterCloseRS AND p_tyBuffer1BffrStat.bBffrMty THEN
//					bRlsMag1	:= TRUE;
//				END_IF
//			END_IF
//
//			IF bNewMag1 = TRUE THEN
//
//				IF p_tyDI.bMag1FixedClampRS = TRUE AND p_tyDI.bMag1RemoteClampRS = TRUE THEN
//					bNewMag1	:= FALSE;
//				END_IF
//
//			ELSIF bRlsMag1 = TRUE THEN
//
//				IF p_tyDI.bMag1FixedUnclampRS = TRUE AND p_tyDI.bMag1RemoteUnclampRS = TRUE AND p_tyDI.bMagConvEntSen1 = TRUE THEN
//					bRlsMag1	:= FALSE;
//				END_IF
//
//			END_IF
//
//		ELSE
//
//			bNewMag1	:= FALSE;
//			bRlsMag1	:= FALSE;
//
//			fbMag1EntrySenOnTm(IN := FALSE);
//
//		END_IF
//
//	END_IF

END_ACTION
```

#### Act_OptP0202_P0003AIVDat.st - not listed in the package file held
```iecst
ACTION Act_OptP0202_P0003AIVDat:

	//Show Change Mag Button only in Manual Exchane Mode
	tyP0202OpsMag1.tyOps.tyBtnChgMag.uiRtStat.0 := p_tyMcParamCurr.eMagExMode = McSetMagXcAutoMode AND p_tyMcParamCurr.eAGVComProtocol <> McSetAGVCommDisabled  OR p_tyNtParamCurr.bProjLifterMagPlatform;;
	tyP0202OpsMag1.tyOps.tyBitmapChgMag.uiRtStat.0 := p_tyMcParamCurr.eMagExMode = McSetMagXcAutoMode AND p_tyMcParamCurr.eAGVComProtocol <> McSetAGVCommDisabled  OR p_tyNtParamCurr.bProjLifterMagPlatform;;
	//LED Wifi
	tyP0202OpsMag1.tyOps.tyBtnAIVWifi.bValue	:= p_bAGVOnline;

	//Change Magazine
	IF p_tyNtParamCurr.bProjBtnInsertRmvMag = TRUE THEN

		IF EDGENEG(p_bOpsStatusRun) THEN
			bNewMag1	:= FALSE;
			tyP0202OpsMag1.tyOps.tyBtnChgMag.bRtLk	:= FALSE;
			tyP0202OpsMag1.tyOps.tyBtnChgMag.bRtCompl	:= FALSE;
			tyP0202OpsMag1.tyOps.tyBtnChgMag.bValue		:= FALSE;
		END_IF

		IF tyP0202OpsMag1.tyOps.tyBtnChgMag.bRtCompl = TRUE THEN
			tyP0202OpsMag1.tyOps.tyBitmapChgMag.usiValueIdx	:= 1;
			tyP0202OpsMag1.tyOps.tyBtnChgMag.bRtLk := TRUE;
			IF 	p_bOpsMagConvLD1NewMagAllw OR p_bOpsMagConvLD1RlsMagAllw OR p_bOpsMagConvLD1RlsMagUmask THEN
				tyP0202OpsMag1.tyOps.tyBtnChgMag.bRtCompl	:= FALSE;
				bNewMag1	:= p_bOpsMagConvLD1NewMagAllw;
				bRlsMag1	:= p_bOpsMagConvLD1RlsMagAllw;
				bEjectMag1  := p_bOpsMagConvLD1ExtMes;
			END_IF
		END_IF

		IF bNewMag1 = TRUE THEN
			tyP0202OpsMag1.tyOps.tyBitmapChgMag.usiValueIdx	:= 1;

			IF p_tyDI.bMag1FixedUnclampRS = FALSE OR p_eMagConv2Clp1Status = Error THEN
				bNewMag1	:= FALSE;
				tyP0202OpsMag1.tyOps.tyBtnChgMag.bValue	:= FALSE;
				tyP0202OpsMag1.tyOps.tyBtnChgMag.bRtLk	:= FALSE;
				tyP0202OpsMag1.tyOps.tyBitmapChgMag.usiValueIdx	:= 0;
			END_IF

		ELSIF bRlsMag1 = TRUE OR bEjectMag1 THEN
				tyP0202OpsMag1.tyOps.tyBitmapChgMag.usiValueIdx	:= 1;
			IF p_tyNtParamCurr.eCustomerReq = Siemens OR p_tyNtParamCurr.eCustomerReq = We_Fabricate THEN
				IF p_bOpsMagConvLD1RlsMagUmask THEN // siemens , read -1 or write TO
					IF p_tyNtParamCurr.eCustomerReq = We_Fabricate THEN
						//bRlsMag1	:= FALSE;
						tyP0202OpsMag1.tyOps.tyBitmapChgMag.usiValueIdx	:= 0;
					END_IF
					tyP0202OpsMag1.tyOps.tyBtnChgMag.bValue	:= FALSE;
					tyP0202OpsMag1.tyOps.tyBtnChgMag.bRtLk	:= FALSE;
				ELSIF p_bOpsMagConvLD1ExtMes THEN //2nd press to eject mag
					bEjectMag1	:= FALSE;
					bRlsMag1	:= FALSE;
					tyP0202OpsMag1.tyOps.tyBtnChgMag.bValue	:= FALSE;
					tyP0202OpsMag1.tyOps.tyBtnChgMag.bRtLk	:= FALSE;
					tyP0202OpsMag1.tyOps.tyBitmapChgMag.usiValueIdx	:= 0;
				ELSIF (p_tyDI.bMag1FixedUnclampRS = TRUE AND p_tyDI.bMagPresentSen1 = FALSE) AND p_tyMcParamCurr.eDSCommA = 0 THEN//smema
					bRlsMag1	:= FALSE;
					tyP0202OpsMag1.tyOps.tyBtnChgMag.bValue	:= FALSE;
					tyP0202OpsMag1.tyOps.tyBtnChgMag.bRtLk	:= FALSE;
					tyP0202OpsMag1.tyOps.tyBitmapChgMag.usiValueIdx	:= 0;
				END_IF

			ELSIF (p_tyDI.bMag1FixedUnclampRS = TRUE AND p_tyDI.bMagPresentSen1 = FALSE)THEN
				bRlsMag1	:= FALSE;
				tyP0202OpsMag1.tyOps.tyBtnChgMag.bValue	:= FALSE;
				tyP0202OpsMag1.tyOps.tyBtnChgMag.bRtLk	:= FALSE;
				tyP0202OpsMag1.tyOps.tyBitmapChgMag.usiValueIdx	:= 0;
			END_IF

		END_IF

		IF p_tyDI.bMagPresentSen1 AND p_tyDI.bMagConvEntSen1 = FALSE THEN
			tyP0202OpsMag1.tyOps.tyBtnChgMag.usiTxtIdx	:= 1;
		ELSE
			tyP0202OpsMag1.tyOps.tyBtnChgMag.usiTxtIdx	:= 0;
			tyP0202OpsMag1.tyOps.tyBtnChgMag.uiMaskRtStat := TRUE;
			IF EDGEPOS(tyP0202OpsMag1.tyOps.tyBtnChgMag.usiTxtIdx =0) THEN
				tyP0202OpsMag1.tyOps.tyBitmapChgMag.usiValueIdx	:= 0;
			END_IF
		END_IF

//		tyP0202OpsMag1.tyOps.tyBtnChgMag.uiMaskRtStat.0	:= p_bOpsMagConvLD1NewMagAllw OR p_bOpsMagConvLD1RlsMagAllw OR p_bOpsMagConvLD1RlsMagUmask;// OR p_tyDI.bInShutterCloseRS;
		tyP0003MMenu.tyMMenuBtn.tyBtnRlsNewMag1.usiTxtIdx := tyP0003MMenu.tyMMenuBtn.tyBtnRlsNewMagBk1.usiTxtIdx + tyP0202OpsMag1.tyOps.tyBtnChgMag.usiTxtIdx;
		tyP0003MMenu.tyMMenuBtn.tyBtnRlsNewMag1.usiTxtIdx := tyP0003MMenu.tyMMenuBtn.tyBtnRlsNewMagBk1.usiTxtIdx + tyP0202OpsMag1.tyOps.tyBtnChgMag.usiTxtIdx;
		tyP0003MMenu.tyMMenuBtn.tyBtnRlsNewMag1.usiBitmapIdx := tyP0003MMenu.tyMMenuBtn.tyBtnRlsNewMagBk1.usiBitmapIdx + 	tyP0202OpsMag1.tyOps.tyBitmapChgMag.usiValueIdx;
		tyP0003MMenu.tyMMenuBtn.tyBtnRlsNewMag1.uiMaskRtStat := tyP0202OpsMag1.tyOps.tyBtnChgMag.uiMaskRtStat ;
	END_IF

END_ACTION
```

#### Act_EntP0203Disp.st
```iecst
ACTION Act_EntP0203Disp:

	//Access Address
	p_tyC0004Navi ACCESS ADR(tyP0203OpsMag2.tyNaviBack);

	p_tyC0005Main ACCESS ADR(tyCommon.tyMain);

	p_tyC0007Notif ACCESS ADR(tyCommon.tyNotif);

	p_tyC0008MsgBox ACCESS ADR(tyP0203OpsMag2.tyMsgBoxHide);

	p_tyC0009Info ACCESS ADR(tyCommon.tyInfo);

	p_tyC0011RcpPopUp ACCESS ADR(tyP0203OpsMag2.tyRcpPopUp);

	p_tyP0203Ops ACCESS ADR(tyP0203OpsMag2.tyOps);
	p_tyP0203IOMonitor ACCESS ADR(tyP0203OpsMag2.tyIOMonitor);
	p_tyP0203BypsInitConv ACCESS ADR(tyP0203OpsMag2.tyBypsInitConv);
	p_tyP0203Param ACCESS ADR(tyP0203OpsMag2.tyParam);

	//Display
	fUIInRtStatHide(ADR(tyP0203OpsMag2.tyIOMonitor.tyLyr.uiRtStat));
	fUIInRtStatHide(ADR(tyP0203OpsMag2.tyParam.tyLyr.uiRtStat));

	tyP0203OpsMag2.tyOps.tyBtnChgParam.uiRtStat.0	:= NOT(p_tyMcParamCurr.bChgParamEn);
	tyP0203OpsMag2.tyParam.tyNumMaxSlt.diValueMax	:= p_tyMagRcpCurrRcp.diTtlSlt;

	IF p_tyNtParamCurr.bMagAutoVerifyPrep = FALSE THEN
		tyP0203OpsMag2.tyIOMonitor.tyBtnMag2FixedClmpRS.usiTxtIdx	:= 75;
		tyP0203OpsMag2.tyIOMonitor.tyBtnMag2FixedUnclmpRS.usiTxtIdx:= 75;
		tyP0203OpsMag2.tyIOMonitor.tyBtnMag2RmtClmpRS.usiTxtIdx	:= 0;
		tyP0203OpsMag2.tyIOMonitor.tyBtnMag2RmtUnclmpRS.usiTxtIdx:= 0;
		tyP0203OpsMag2.tyIOMonitor.tyBtnMag2FixedClampCtrl.usiTxtIdx:= 41;
		tyP0203OpsMag2.tyIOMonitor.tyBtnMag2RemoteClampCtrl.usiTxtIdx:= 18;
	ELSE
		tyP0203OpsMag2.tyIOMonitor.tyBtnMag2FixedClmpRS.usiTxtIdx	:= 75;
		tyP0203OpsMag2.tyIOMonitor.tyBtnMag2FixedUnclmpRS.usiTxtIdx:= 75;
		tyP0203OpsMag2.tyIOMonitor.tyBtnMag2RmtClmpRS.usiTxtIdx	:= 0;
		tyP0203OpsMag2.tyIOMonitor.tyBtnMag2RmtUnclmpRS.usiTxtIdx:= 0;
		tyP0203OpsMag2.tyIOMonitor.tyBtnMag2FixedClampCtrl.usiTxtIdx:= 41;
		tyP0203OpsMag2.tyIOMonitor.tyBtnMag2RemoteClampCtrl.usiTxtIdx:= 18;

	END_IF

	fUIInRtStatHide(ADR(tyP0203OpsMag2.tyOps.tyBtnAIVWifi.uiRtStat));
	fUIInRtStatHide(ADR(tyP0203OpsMag2.tyOps.tyTxtLblAIV.uiRtStat));

	tyP0203OpsMag2.tyParam.tyNumMaxSlt.diValueMax	:= p_tyMagRcpCurrRcp.diTtlSlt;

END_ACTION
```

#### Act_OptP0203UpdtDat.st
```iecst
ACTION Act_OptP0203UpdtDat:

	//Status
	fbMcStatUpdtTm(IN := TRUE);
	IF fbMcStatUpdtTm.Q = TRUE THEN
		fbMcStatUpdtTm(IN := FALSE);

		IF p_tyNtParamCurr.bProjLifterMagPlatform THEN
			tyP0203OpsMag2.tyOps.tyStringMcStat.sValue	:= p_sOpsLifMagLDStepTxt;
		ELSE
			tyP0203OpsMag2.tyOps.tyStringMcStat.sValue	:= p_sOpsMagConvLD2StepTxt;
		END_IF

	END_IF

	//Mode
	tyP0203OpsMag2.tyOps.tyTxtMod.usiValueIdx	:= p_tyProdRcpCurrRcp1.usiMcMod;

	//Width
	IF p_tyNtParamCurr.bAWPrep = TRUE AND p_tyMcParamCurr.bAWDis = FALSE THEN
		tyP0203OpsMag2.tyOps.tyNumWidth.diValue	:= p_tyMcParamCurr.diWidthAtHmPosInUM - p_diAWOpenActualPos;
		tyP0203OpsMag2.tyOps.tyNumWidth2.diValue	:= p_tyMcParamCurr.diWidthAtHmPosInUM - p_diAWOpenActualPos;
	ELSE
		tyP0203OpsMag2.tyOps.tyNumWidth.diValue	:= p_tyProdRcpCurrRcp1.diWidthInUM;
		tyP0203OpsMag2.tyOps.tyNumWidth2.diValue	:= p_tyProdRcpCurrRcp1.diWidthInUM2;
	END_IF

	//Program Info
	IF p_tyNtParamCurr.eProjMag <> LDMagQuadruple THEN
		IF p_tyNtParamCurr.bProjAutoRcpPrep AND p_tyMcParamCurr.bHermesSvyEn THEN
			tyP0203OpsMag2.tyOps.tyNumMinSltRange.diValue		:= p_diLinkAutoRcpMag2MinSlt;
			tyP0203OpsMag2.tyOps.tyNumMaxSltRange.diValue		:= p_diLinkAutoRcpMag2MaxSlt;
			tyP0203OpsMag2.tyOps.tyNumPitch.diValue				:= p_diLinkAutoRcpMag2Pitch;
			tyP0203OpsMag2.tyOps.tyStringProdNm.sValue			:= p_tyAutoRcpMagRcp[2].sWorkOrderId;
		ELSE
			tyP0203OpsMag2.tyOps.tyNumMinSltRange.diValue		:= p_tyProdRcpCurrRcp2.diMinSltValue;
			tyP0203OpsMag2.tyOps.tyNumMaxSltRange.diValue		:= p_tyProdRcpCurrRcp2.diMaxSltValue;
			tyP0203OpsMag2.tyOps.tyNumPitch.diValue				:= p_tyProdRcpCurrRcp2.diPitch;
			tyP0203OpsMag2.tyOps.tyStringProdNm.sValue			:= p_tyProdRcpCurrRcp2.sRcpNm;
		END_IF
		tyP0203OpsMag2.tyOps.tyBtnToptoBtm.bValue			:= p_tyProdRcpCurrRcp2.bTopToBtm;
		//Magazine Info
		tyP0203OpsMag2.tyOps.tyStringMagNm.sValue	:= p_tyMagRcpCurrRcp.sRcpNm;
	ELSE
		CASE p_tyProdRcpCurrRcp2.usiMcMod OF
			0,2:
				tyP0203OpsMag2.tyOps.tyStringProdNm.sValue		:= p_tyProdRcpCurrRcp2.sRcpNm;
				tyP0203OpsMag2.tyOps.tyNumMinSltRange.diValue		:= p_tyProdRcpCurrRcp2.diMinSltValue;
				tyP0203OpsMag2.tyOps.tyNumMaxSltRange.diValue		:= p_tyProdRcpCurrRcp2.diMaxSltValue;
				tyP0203OpsMag2.tyOps.tyBtnToptoBtm.bValue			:= p_tyProdRcpCurrRcp2.bTopToBtm;
				tyP0203OpsMag2.tyOps.tyNumPitch.diValue			:= p_tyProdRcpCurrRcp2.diPitch;
				//Magazine Info
				tyP0203OpsMag2.tyOps.tyStringMagNm.sValue	:= p_tyMagRcpCurrRcp.sRcpNm;
			1:

				tyP0203OpsMag2.tyOps.tyStringProdNm.sValue		:= p_tyProdRcpCurrRcp2.sRcpNm;
				tyP0203OpsMag2.tyOps.tyNumMinSltRange.diValue		:= p_tyProdRcpCurrRcp2.diMinSltValueRear;
				tyP0203OpsMag2.tyOps.tyNumMaxSltRange.diValue		:= p_tyProdRcpCurrRcp2.diMaxSltValueRear;
				tyP0203OpsMag2.tyOps.tyBtnToptoBtm.bValue			:= p_tyProdRcpCurrRcp2.bTopToBtm;
				tyP0203OpsMag2.tyOps.tyNumPitch.diValue			:= p_tyProdRcpCurrRcp2.diPitchRear;
				//Magazine Info
				tyP0203OpsMag2.tyOps.tyStringMagNm.sValue	:= p_tyMagRcpCurrRcp1.sRcpNm;
		END_CASE
	END_IF

	//Magazine Info
//	tyP0203OpsMag2.tyOps.tyStringMagNm.sValue	:= p_tyMagRcpCurrRcp.sRcpNm;

	IF p_bBuffer2MagPresent = TRUE THEN
		tyP0203OpsMag2.tyOps.tyNumMag2AvlQty.diValue	:= p_tyBuffer2BffrStat.diTtlGdBrd + p_tyBuffer2BffrStat.diTtlBadBrd;
		tyP0203OpsMag2.tyOps.tyNumMag2TtlSlt.diValue	:= p_tyBuffer2BffrStat.diTtlBrdCap;
	ELSE
		tyP0203OpsMag2.tyOps.tyNumMag2AvlQty.diValue	:= 0;
		tyP0203OpsMag2.tyOps.tyNumMag2TtlSlt.diValue	:= 0;
	END_IF

	//Magazine Present States
	IF p_bBuffer2MagPresent = TRUE THEN

		IF p_tyBuffer2BffrStat.bBffrFull = TRUE THEN
			tyP0203OpsMag2.tyOps.tyTxtMag2Stat.usiValueIdx := 2;
			tyP0203OpsMag2.tyOps.tyTxtMag2Stat.usiColor	   := 0;
		ELSIF p_tyBuffer2BffrStat.bBffrMty = TRUE THEN
			tyP0203OpsMag2.tyOps.tyTxtMag2Stat.usiValueIdx := 1;
			tyP0203OpsMag2.tyOps.tyTxtMag2Stat.usiColor	   := 1;
		ELSE
			tyP0203OpsMag2.tyOps.tyTxtMag2Stat.usiValueIdx := 3;
			tyP0203OpsMag2.tyOps.tyTxtMag2Stat.usiColor	   := 0;
		END_IF

	ELSE
		tyP0203OpsMag2.tyOps.tyTxtMag2Stat.usiValueIdx := 0;
		tyP0203OpsMag2.tyOps.tyTxtMag2Stat.usiColor	   := 1;
	END_IF

	//Product Recipe 254
	tyP0203OpsMag2.tyOps.tyHotspotShowLRcp.uiRtStat.0 := NOT(tyP0203OpsMag2.tyOps.tyStringProdNm.sValue <> '');

	IF tyP0203OpsMag2.tyOps.tyHotspotShowLRcp.bRtCompl = TRUE THEN
		tyP0203OpsMag2.tyOps.tyHotspotShowLRcp.bRtCompl := FALSE;

		fUIInRtStatOff(ADR(tyP0203OpsMag2.tyRcpPopUp.tyLyr.uiRtStat));

		tyP0203OpsMag2.tyRcpPopUp.tyStringInfo.sValue  := p_tyProdRcpCurrRcp1.sRcpNm;

	ELSIF tyP0203OpsMag2.tyRcpPopUp.tyHotspotClose.bRtCompl = TRUE THEN
		tyP0203OpsMag2.tyRcpPopUp.tyHotspotClose.bRtCompl := FALSE;

		fUIInRtStatHide(ADR(tyP0203OpsMag2.tyRcpPopUp.tyLyr.uiRtStat));

	END_IF
END_ACTION
```

#### Act_OptP0203IOMonitor.st
```iecst
ACTION Act_OptP0203IOMonitor:

	IF tyP0203OpsMag2.tyOps.tyHotspotIOMonitor.bRtCompl = TRUE THEN
		tyP0203OpsMag2.tyOps.tyHotspotIOMonitor.bRtCompl	:= FALSE;

		fUIInRtStatOff(ADR(tyP0203OpsMag2.tyIOMonitor.tyLyr.uiRtStat));

		p_tyC0004Navi ACCESS ADR(tyP0203OpsMag2.tyNaviHide);

	ELSIF tyP0203OpsMag2.tyIOMonitor.tyHotspotClose.bRtCompl = TRUE THEN
		tyP0203OpsMag2.tyIOMonitor.tyHotspotClose.bRtCompl	:= FALSE;

		fUIInRtStatHide(ADR(tyP0203OpsMag2.tyIOMonitor.tyLyr.uiRtStat));

		p_tyC0004Navi ACCESS ADR(tyP0203OpsMag2.tyNaviBack);

	END_IF

	IF tyP0203OpsMag2.tyIOMonitor.tyLyr.uiRtStat.0 = FALSE THEN

		//Digital Input
		tyP0203OpsMag2.tyIOMonitor.tyBtnSafetyRlySig.bValue				:= p_tyDI.bSafetyRlySig;
		tyP0203OpsMag2.tyIOMonitor.tyBtnEStop.bValue					:= p_tyDI.bEStopSig;
		tyP0203OpsMag2.tyIOMonitor.tyBtnCoverSWSig.bValue				:= p_tyDI.bCoverSWSig;
		tyP0203OpsMag2.tyIOMonitor.tyBtnDSBA.bValue						:= p_tyDI.bDSBA;
		tyP0203OpsMag2.tyIOMonitor.tyBtnDSBB.bValue						:= p_tyDI.bDSBB;
		tyP0203OpsMag2.tyIOMonitor.tyBtnMag2FixedClmpRS.bValue			:= p_tyDI.bMag2FixedClampRS;
		tyP0203OpsMag2.tyIOMonitor.tyBtnMag2FixedUnclmpRS.bValue		:= p_tyDI.bMag2FixedUnclampRS;
		tyP0203OpsMag2.tyIOMonitor.tyBtnMag2RmtClmpRS.bValue			:= p_tyDI.bMag2RemoteClampRS;
		tyP0203OpsMag2.tyIOMonitor.tyBtnMag2RmtUnclmpRS.bValue			:= p_tyDI.bMag2RemoteUnclampRS;
		tyP0203OpsMag2.tyIOMonitor.tyBtnMag2ConvEntrySen.bValue			:= p_tyDI.bMagConvEntSen2;
		tyP0203OpsMag2.tyIOMonitor.tyBtnMag2PresentSen.bValue			:= p_tyDI.bMagPresentSen2;
		tyP0203OpsMag2.tyIOMonitor.tyBtnMag2AIVInPosSen1.bValue			:= p_tyDI.bMag2AGVInPosSen1;
		tyP0203OpsMag2.tyIOMonitor.tyBtnMag2AIVInPosSen2.bValue			:= p_tyDI.bMag2AGVInPosSen2;
		tyP0203OpsMag2.tyIOMonitor.tyBtnMag2OrientationChkSen1.bValue	:= p_tyDI.bMag2OrientChkSen1;
		tyP0203OpsMag2.tyIOMonitor.tyBtnMag2OrientationChkSen2.bValue	:= p_tyDI.bMag2OrientChkSen2;

		tyP0203OpsMag2.tyIOMonitor.tyBtnSelUnclampRS.bValue				:= p_tyDI.bMag2SelUnClampRS;

		tyP0203OpsMag2.tyIOMonitor.tyBtnCAB717Sen.bValue				:= p_tyDI.bMagConvCAB717MagSen2;
		tyP0203OpsMag2.tyIOMonitor.tyBtnHeightSen.bValue				:= p_tyDI.bMagConvHeightSen2 OR p_tyDI.bHighMagDetSen2;
		tyP0203OpsMag2.tyIOMonitor.tyBtnMagSmallSen.bValue				:= p_tyDI.bMagConvSmallMagSen2;
		tyP0203OpsMag2.tyIOMonitor.tyBtnMagLargeSen.bValue				:= p_tyDI.bMagConvLargeMagSen2;
		tyP0203OpsMag2.tyIOMonitor.tyBtnMagDetSen.bValue				:= p_tyDI.bMag2FixedSideDetect;
		tyP0203OpsMag2.tyIOMonitor.tyBtnTrllyExtRS.bValue				:= p_tyDI.bTrolleyExtRS2;
		tyP0203OpsMag2.tyIOMonitor.tyBtnTrllyPresentSen.bValue			:= p_tyDI.bTrolleyPreSen2;
		tyP0203OpsMag2.tyIOMonitor.tyBtnSltLckSen.bValue				:= p_tyDI.bSlotLckSenMag2;

		//Digital Output
		tyP0203OpsMag2.tyIOMonitor.tyBtnSafetyRlyRst.bValue				:= p_tyDO.bSafetyRlyRst;
		tyP0203OpsMag2.tyIOMonitor.tyBtnTLGreen.bValue					:= p_tyDO.bTLGreen;
		tyP0203OpsMag2.tyIOMonitor.tyBtnTLAmber.bValue					:= p_tyDO.bTLAmber;
		tyP0203OpsMag2.tyIOMonitor.tyBtnTLRed.bValue					:= p_tyDO.bTLRed;
		tyP0203OpsMag2.tyIOMonitor.tyBtnBuzzer.bValue					:= p_tyDO.bBuzzer;
		tyP0203OpsMag2.tyIOMonitor.tyBtnDBAA.bValue						:= p_tyDO.bDBAA;
		tyP0203OpsMag2.tyIOMonitor.tyBtnDBAB.bValue						:= p_tyDO.bDBAB;
		tyP0203OpsMag2.tyIOMonitor.tyBtnMag2FixedClampCtrl.bValue		:= p_tyDO.bMag2FixedClampCtrl;
		tyP0203OpsMag2.tyIOMonitor.tyBtnMag2RemoteClampCtrl.bValue		:= p_tyDO.bMag2RemoteClampCtrl;
		tyP0203OpsMag2.tyIOMonitor.tyBtnMag2ConvMtrIn.bValue			:= p_tyDO.bMag2ConvMtrIn;
		tyP0203OpsMag2.tyIOMonitor.tyBtnMag2ConvMtrOut.bValue			:= p_tyDO.bMag2ConvMtrOut;
		tyP0203OpsMag2.tyIOMonitor.tyBtnMagSelClampCtrl.bValue			:= p_tyDO.bMag2SelClampCtrl;
		tyP0203OpsMag2.tyIOMonitor.tyBtnTrllyExtCtrl.bValue				:= p_tyDO.bTrolleyLckCtrl2;
	END_IF

END_ACTION
```

#### Act_OptP0203AIVDat.st
```iecst
ACTION Act_OptP0203AIVDat:

	//Show Change Mag Button only in Manual Exchane Mode
	tyP0203OpsMag2.tyOps.tyBtnChgMag.uiRtStat.0 := p_tyMcParamCurr.eMagExMode = McSetMagXcAutoMode AND p_tyMcParamCurr.eAGVComProtocol <> McSetAGVCommDisabled OR p_tyNtParamCurr.bProjLifterMagPlatform;;
	tyP0203OpsMag2.tyOps.tyBitmapChgMag.uiRtStat.0 := p_tyMcParamCurr.eMagExMode = McSetMagXcAutoMode AND p_tyMcParamCurr.eAGVComProtocol <> McSetAGVCommDisabled OR p_tyNtParamCurr.bProjLifterMagPlatform;;
	//LED Wifi
	tyP0203OpsMag2.tyOps.tyBtnAIVWifi.bValue	:= p_bAGVOnline;

	//Change Magazine
	IF p_tyNtParamCurr.bProjBtnInsertRmvMag = TRUE THEN

		IF EDGENEG(p_bOpsStatusRun) THEN
			bNewMag2	:= FALSE;
			tyP0203OpsMag2.tyOps.tyBtnChgMag.bRtLk	:= FALSE;
			tyP0203OpsMag2.tyOps.tyBtnChgMag.bRtCompl	:= FALSE;
			tyP0203OpsMag2.tyOps.tyBtnChgMag.bValue		:= FALSE;
		END_IF

		IF tyP0203OpsMag2.tyOps.tyBtnChgMag.bRtCompl = TRUE THEN
			tyP0203OpsMag2.tyOps.tyBitmapChgMag.usiValueIdx	:= 1;
			tyP0203OpsMag2.tyOps.tyBtnChgMag.bRtLk	:= TRUE;
			IF 	p_bOpsMagConvLD2NewMagAllw OR p_bOpsMagConvLD2RlsMagAllw OR p_bOpsMagConvLD2RlsMagUmask THEN
				tyP0203OpsMag2.tyOps.tyBtnChgMag.bRtCompl	:= FALSE;
				bNewMag2	:= p_bOpsMagConvLD2NewMagAllw;
				bRlsMag2	:= p_bOpsMagConvLD2RlsMagAllw;
				bEjectMag2  := p_bOpsMagConvLD2ExtMes;
			END_IF
		END_IF

		IF bNewMag2 = TRUE THEN
			tyP0203OpsMag2.tyOps.tyBitmapChgMag.usiValueIdx	:= 1;
			IF p_tyDI.bMag2FixedUnclampRS = FALSE OR p_eMagConv2Clp2Status = Error  THEN
				bNewMag2	:= FALSE;
				tyP0203OpsMag2.tyOps.tyBtnChgMag.bValue	:= FALSE;
				tyP0203OpsMag2.tyOps.tyBtnChgMag.bRtLk	:= FALSE;
				tyP0203OpsMag2.tyOps.tyBitmapChgMag.usiValueIdx	:= 0;
			END_IF

		ELSIF bRlsMag2 = TRUE OR bEjectMag2 THEN
			tyP0203OpsMag2.tyOps.tyBitmapChgMag.usiValueIdx	:= 1;
			IF p_tyNtParamCurr.eCustomerReq = Siemens OR p_tyNtParamCurr.eCustomerReq = We_Fabricate THEN
				IF p_bOpsMagConvLD2RlsMagUmask THEN // siemens , read -1 or write TO
					IF p_tyNtParamCurr.eCustomerReq = We_Fabricate THEN
						//bRlsMag2	:= FALSE;
						tyP0203OpsMag2.tyOps.tyBitmapChgMag.usiValueIdx	:= 0;
					END_IF
					tyP0203OpsMag2.tyOps.tyBtnChgMag.bValue	:= FALSE;
					tyP0203OpsMag2.tyOps.tyBtnChgMag.bRtLk	:= FALSE;
				ELSIF p_bOpsMagConvLD2ExtMes THEN //2nd press to eject mag
					bEjectMag2	:= FALSE;
					bRlsMag2	:= FALSE;
					tyP0203OpsMag2.tyOps.tyBtnChgMag.bValue	:= FALSE;
					tyP0203OpsMag2.tyOps.tyBtnChgMag.bRtLk	:= FALSE;
					tyP0203OpsMag2.tyOps.tyBitmapChgMag.usiValueIdx	:= 0;
				ELSIF (p_tyDI.bMag2FixedUnclampRS = TRUE AND p_tyDI.bMagPresentSen2 = FALSE) AND p_tyMcParamCurr.eDSCommA = 0 THEN//smema
					bRlsMag2	:= FALSE;
					tyP0203OpsMag2.tyOps.tyBtnChgMag.bValue	:= FALSE;
					tyP0203OpsMag2.tyOps.tyBtnChgMag.bRtLk	:= FALSE;
					tyP0203OpsMag2.tyOps.tyBitmapChgMag.usiValueIdx	:= 0;
				END_IF

			ELSIF (p_tyDI.bMag2FixedUnclampRS = TRUE AND p_tyDI.bMagPresentSen2 = FALSE) THEN
				bRlsMag2	:= FALSE;
				tyP0203OpsMag2.tyOps.tyBtnChgMag.bValue	:= FALSE;
				tyP0203OpsMag2.tyOps.tyBtnChgMag.bRtLk	:= FALSE;
				tyP0203OpsMag2.tyOps.tyBitmapChgMag.usiValueIdx	:= 0;
			END_IF

		END_IF

		IF p_tyDI.bMagPresentSen2 AND p_tyDI.bMagConvEntSen2 = FALSE THEN
			tyP0203OpsMag2.tyOps.tyBtnChgMag.usiTxtIdx	:= 1;
		ELSE
			tyP0203OpsMag2.tyOps.tyBtnChgMag.usiTxtIdx	:= 0;
			tyP0203OpsMag2.tyOps.tyBtnChgMag.uiMaskRtStat := TRUE;
			IF EDGEPOS(tyP0203OpsMag2.tyOps.tyBtnChgMag.usiTxtIdx =0) THEN
				tyP0203OpsMag2.tyOps.tyBitmapChgMag.usiValueIdx	:= 0;
			END_IF
		END_IF

	//	tyP0203OpsMag2.tyOps.tyBtnChgMag.uiMaskRtStat.0	:= p_bOpsMagConvLD2NewMagAllw OR p_bOpsMagConvLD2RlsMagAllw OR p_bOpsMagConvLD2RlsMagUmask;// OR p_tyDI.bInShutterCloseRS;

	END_IF
END_ACTION
```

#### Act_OptP0203ChgParam.st
```iecst
ACTION Act_OptP0203ChgParam:

	tyP0203OpsMag2.tyParam.tyNumMinSlt.diValueMax		:= tyP0203OpsMag2.tyParam.tyNumMaxSlt.diValue;
	tyP0203OpsMag2.tyParam.tyNumMaxSlt.diValueMin		:= tyP0203OpsMag2.tyParam.tyNumMinSlt.diValue;
	tyP0203OpsMag2.tyParam.tyNumPitch.diValueMax		:= tyP0203OpsMag2.tyParam.tyNumMaxSlt.diValue - tyP0203OpsMag2.tyParam.tyNumMinSlt.diValue + 1;
	tyP0203OpsMag2.tyParam.tyNumPitch.diValueMin		:= 1;

	tyP0203OpsMag2.tyParam.tyNumMinSltRear.diValueMax		:= tyP0203OpsMag2.tyParam.tyNumMaxSltRear.diValue;
	tyP0203OpsMag2.tyParam.tyNumMaxSltRear.diValueMin		:= tyP0203OpsMag2.tyParam.tyNumMinSltRear.diValue;
	tyP0203OpsMag2.tyParam.tyNumPitchRear.diValueMax		:= tyP0203OpsMag2.tyParam.tyNumMaxSltRear.diValue - tyP0203OpsMag2.tyParam.tyNumMinSltRear.diValue + 1;
	tyP0203OpsMag2.tyParam.tyNumPitchRear.diValueMin		:= 1;

	tyP0203OpsMag2.tyParam.tyNumMtrPshrExtSpd.diValueMin	:= p_tyNtParamCurr.tyProdRcpMtrPshrExtSpd.diMin;
	tyP0203OpsMag2.tyParam.tyNumMtrPshrExtSpd.diValueMax	:= p_tyNtParamCurr.tyProdRcpMtrPshrExtSpd.diMax;
	tyP0203OpsMag2.tyParam.tyNumMtrPshrExtTorq.diValueMin	:= p_tyNtParamCurr.tyProdRcpMtrPshrExtTorq.diMin;
	tyP0203OpsMag2.tyParam.tyNumMtrPshrExtTorq.diValueMax	:= p_tyNtParamCurr.tyProdRcpMtrPshrExtTorq.diMax;
	tyP0203OpsMag2.tyParam.tyNumPshrOffset.diValueMin		:= -(p_tyProdRcpCurrRcp2.diWidthInUM/2-p_tyMcParamCurr.diAWPusherAtHmPosInUM-5000 );
	tyP0203OpsMag2.tyParam.tyNumPshrOffset.diValueMax		:= (p_tyProdRcpCurrRcp2.diWidthInUM/2-p_tyMcParamCurr.diAWPusherAtHmPosInUM-5000 );

	//Control
	IF tyP0203OpsMag2.tyOps.tyBtnChgParam.bRtCompl = TRUE THEN
		tyP0203OpsMag2.tyOps.tyBtnChgParam.bRtCompl	:= FALSE;

		tyProdRcpCurrRcpWr	:= p_tyProdRcpCurrRcp0;

		tyP0203OpsMag2.tyParam.tyDrpDnMcMode.usiValueIdx	:= p_tyProdRcpCurrRcp0.usiMcMod;
		tyP0203OpsMag2.tyParam.tyNumMinSlt.diValue	:= p_tyProdRcpCurrRcp0.diMinSltValue;
		tyP0203OpsMag2.tyParam.tyNumMaxSlt.diValue	:= p_tyProdRcpCurrRcp0.diMaxSltValue;
		tyP0203OpsMag2.tyParam.tyNumPitch.diValue		:= p_tyProdRcpCurrRcp0.diPitch;

		tyP0203OpsMag2.tyParam.tyNumMinSltRear.diValue	:= p_tyProdRcpCurrRcp0.diMinSltValueRear;
		tyP0203OpsMag2.tyParam.tyNumMaxSltRear.diValue	:= p_tyProdRcpCurrRcp0.diMaxSltValueRear;
		tyP0203OpsMag2.tyParam.tyNumPitchRear.diValue		:= p_tyProdRcpCurrRcp0.diPitchRear;

		tyP0203OpsMag2.tyParam.tyNumMtrPshrExtSpd.diValue		:= p_tyProdRcpCurrRcp0.diMtrPshrExtSpd;
		tyP0203OpsMag2.tyParam.tyNumMtrPshrExtTorq.diValue	:= p_tyProdRcpCurrRcp0.diMtrPshrExtTorq;
		tyP0203OpsMag2.tyParam.tyNumPshrOffset.diValue		:= p_tyProdRcpCurrRcp0.diPshrOffset;

		fUIInRtStatOff(ADR(tyP0203OpsMag2.tyParam.tyLyr.uiRtStat));

	END_IF

	tyP0203OpsMag2.tyOps.tyBtnChgParam.bValue		:= tyP0203OpsMag2.tyParam.tyLyr.uiRtStat.0 = FALSE;

	IF tyP0203OpsMag2.tyParam.tyLyr.uiRtStat.0 = FALSE THEN

		IF tyP0203OpsMag2.tyParam.tyBtnSave.bRtCompl = TRUE THEN

			tyProdRcpCurrRcpWr.usiMcMod	:= tyP0203OpsMag2.tyParam.tyDrpDnMcMode.usiValueIdx;
			tyProdRcpCurrRcpWr.diMinSltValue := tyP0203OpsMag2.tyParam.tyNumMinSlt.diValue;
			tyProdRcpCurrRcpWr.diMaxSltValue := tyP0203OpsMag2.tyParam.tyNumMaxSlt.diValue;
			tyProdRcpCurrRcpWr.diPitch := tyP0203OpsMag2.tyParam.tyNumPitch.diValue;

			tyProdRcpCurrRcpWr.diMinSltValueRear := tyP0203OpsMag2.tyParam.tyNumMinSltRear.diValue;
			tyProdRcpCurrRcpWr.diMaxSltValueRear := tyP0203OpsMag2.tyParam.tyNumMaxSltRear.diValue;
			tyProdRcpCurrRcpWr.diPitchRear := tyP0203OpsMag2.tyParam.tyNumPitchRear.diValue;

			tyProdRcpCurrRcpWr.diMtrPshrExtSpd := tyP0203OpsMag2.tyParam.tyNumMtrPshrExtSpd.diValue;
			tyProdRcpCurrRcpWr.diMtrPshrExtTorq := tyP0203OpsMag2.tyParam.tyNumMtrPshrExtTorq.diValue;
			tyProdRcpCurrRcpWr.diPshrOffset := tyP0203OpsMag2.tyParam.tyNumPshrOffset.diValue;

			eProdRcpAct	:= ProdRcpActWriteCurrRcpParam;

			IF p_eProdRcpStatus = Done AND p_eProdRcpStat = ProdRcpActWriteCurrRcpParam THEN
				eProdRcpAct	:= ProdRcpActIdle;

				//UIP0400
				tyP0400ProdSel.tyProdSel.tyTxtMcMode.usiValueIdx	:= p_tyProdRcpCurrRcp0.usiMcMod;

				tyP0400ProdSel.tyProdSel.tyNumMinSlt.diValue	:= p_tyProdRcpCurrRcp0.diMinSltValue;
				tyP0400ProdSel.tyProdSel.tyNumMaxSlt.diValue	:= p_tyProdRcpCurrRcp0.diMaxSltValue;
				tyP0400ProdSel.tyProdSel.tyNumPitch.diValue		:= p_tyProdRcpCurrRcp0.diPitch;

				tyP0400ProdSel.tyProdSel.tyNumMinSltRear.diValue	:= p_tyProdRcpCurrRcp0.diMinSltValueRear;
				tyP0400ProdSel.tyProdSel.tyNumMaxSltRear.diValue	:= p_tyProdRcpCurrRcp0.diMaxSltValueRear;
				tyP0400ProdSel.tyProdSel.tyNumPitchRear.diValue		:= p_tyProdRcpCurrRcp0.diPitchRear;

				tyP0400ProdSel.tyProdSel.tyNumMtrPshrExtSpd.diValue		:= p_tyProdRcpCurrRcp0.diMtrPshrExtSpd;
				tyP0400ProdSel.tyProdSel.tyNumMtrPshrExtTorq.diValue	:= p_tyProdRcpCurrRcp0.diMtrPshrExtTorq;
				tyP0400ProdSel.tyProdSel.tyNumPshrOffset.diValue		:= p_tyProdRcpCurrRcp0.diPshrOffset;

				tyP0203OpsMag2.tyParam.tyBtnSave.bRtCompl			:= FALSE;
				tyP0203OpsMag2.tyParam.tyBtnSave.bValue				:= FALSE;

				fUIInRtStatHide(ADR(tyP0203OpsMag2.tyParam.tyLyr.uiRtStat));

			ELSIF p_eProdRcpStatus = Error THEN
				p_tyC0008MsgBox ACCESS ADR(tyP0203OpsMag2.tyMsgBoxSaveErr);

				IF tyP0203OpsMag2.tyMsgBoxSaveErr.tyBtnNo.bRtCompl = TRUE THEN
					tyP0203OpsMag2.tyMsgBoxSaveErr.tyBtnNo.bRtCompl	:= FALSE;
					tyP0203OpsMag2.tyMsgBoxSaveErr.tyBtnNo.bValue	:= FALSE;

					p_tyC0008MsgBox ACCESS ADR(tyP0203OpsMag2.tyMsgBoxHide);

					//Restore Param
					tyProdRcpCurrRcpWr	:= p_tyProdRcpCurrRcp2;

					tyP0203OpsMag2.tyParam.tyBtnSave.bRtCompl		:= FALSE;
					tyP0203OpsMag2.tyParam.tyBtnSave.bValue			:= FALSE;

					fUIInRtStatHide(ADR(tyP0203OpsMag2.tyParam.tyLyr.uiRtStat));

				END_IF

			END_IF

		ELSIF tyP0203OpsMag2.tyParam.tyBtnCancel.bRtCompl = TRUE THEN
			tyP0203OpsMag2.tyParam.tyBtnCancel.bRtCompl				:= FALSE;
			tyP0203OpsMag2.tyParam.tyBtnCancel.bValue				:= FALSE;

			fUIInRtStatHide(ADR(tyP0203OpsMag2.tyParam.tyLyr.uiRtStat));

		END_IF

	END_IF

	//Mask
	tyP0203OpsMag2.tyOps.tyBtnChgParam.uiMaskRtStat.0	:= p_tyUsrMgmtCurrAccessRgt.bChgParam AND p_bOpsStatusStop;

END_ACTION
```

#### Act_OptP0203InsertRmvMag.st
```iecst
ACTION Act_OptP0203InsertRmvMag:

	//Insert & Removed Magazine Manually Without Button Control
//	IF p_tyNtParamCurr.bProjBtnInsertRmvMag = FALSE THEN
//
//		IF p_bOpsStatusRun AND p_bOpsMagConvLD2InitDone THEN
//
//			fbMag2EntrySenOnTm(IN := p_tyDI.bMagPresentSen2 OR p_tyDI.bMagConvEntSen2);
//
//			IF bNewMag2 = FALSE AND bRlsMag2 = FALSE THEN
//				IF p_bOpsMagConvLD2NewMagAllw AND fbMag2EntrySenOnTm.Q AND NOT p_bOpsMagConvLD2MagExitedWait THEN
//					bNewMag2	:= TRUE;
//				END_IF
//
//				IF p_bOpsMagConvLD2RlsMagAllw AND p_tyDI.bMagPresentSen2 AND p_tyDI.bInShutterCloseRS AND p_tyBuffer2BffrStat.bBffrMty THEN
//					bRlsMag2	:= TRUE;
//				END_IF
//			END_IF
//
//			IF bNewMag2 = TRUE THEN
//
//				IF p_tyDI.bMag2FixedClampRS = TRUE AND p_tyDI.bMag2RemoteClampRS THEN
//					bNewMag2	:= FALSE;
//				END_IF
//
//			ELSIF bRlsMag2 = TRUE THEN
//
//				IF p_tyDI.bMag2FixedUnclampRS = TRUE AND p_tyDI.bMag2RemoteUnclampRS = TRUE AND p_tyDI.bMagConvEntSen2 = TRUE THEN
//					bRlsMag2	:= FALSE;
//				END_IF
//
//			END_IF
//
//		ELSE
//
//			bNewMag2	:= FALSE;
//			bRlsMag2	:= FALSE;
//
//			fbMag2EntrySenOnTm(IN := FALSE);
//
//		END_IF
//
//	END_IF

END_ACTION
```

#### Act_OptP0203_P0003AIVDat.st - not listed in the package file held
```iecst
ACTION Act_OptP0203_P0003AIVDat:

	//Show Change Mag Button only in Manual Exchane Mode
	tyP0203OpsMag2.tyOps.tyBtnChgMag.uiRtStat.0 := p_tyMcParamCurr.eMagExMode = McSetMagXcAutoMode AND p_tyMcParamCurr.eAGVComProtocol <> McSetAGVCommDisabled OR p_tyNtParamCurr.bProjLifterMagPlatform;;
	tyP0203OpsMag2.tyOps.tyBitmapChgMag.uiRtStat.0 := p_tyMcParamCurr.eMagExMode = McSetMagXcAutoMode AND p_tyMcParamCurr.eAGVComProtocol <> McSetAGVCommDisabled OR p_tyNtParamCurr.bProjLifterMagPlatform;;
	//LED Wifi
	tyP0203OpsMag2.tyOps.tyBtnAIVWifi.bValue	:= p_bAGVOnline;

	//Change Magazine
	IF p_tyNtParamCurr.bProjBtnInsertRmvMag = TRUE THEN

		IF EDGENEG(p_bOpsStatusRun) THEN
			bNewMag2	:= FALSE;
			tyP0203OpsMag2.tyOps.tyBtnChgMag.bRtLk	:= FALSE;
			tyP0203OpsMag2.tyOps.tyBtnChgMag.bRtCompl	:= FALSE;
			tyP0203OpsMag2.tyOps.tyBtnChgMag.bValue		:= FALSE;
		END_IF

		IF tyP0203OpsMag2.tyOps.tyBtnChgMag.bRtCompl = TRUE THEN
			tyP0203OpsMag2.tyOps.tyBitmapChgMag.usiValueIdx	:= 1;
			tyP0203OpsMag2.tyOps.tyBtnChgMag.bRtLk	:= TRUE;
			IF 	p_bOpsMagConvLD2NewMagAllw OR p_bOpsMagConvLD2RlsMagAllw OR p_bOpsMagConvLD2RlsMagUmask THEN
				tyP0203OpsMag2.tyOps.tyBtnChgMag.bRtCompl	:= FALSE;
				bNewMag2	:= p_bOpsMagConvLD2NewMagAllw;
				bRlsMag2	:= p_bOpsMagConvLD2RlsMagAllw;
				bEjectMag2  := p_bOpsMagConvLD2ExtMes;
			END_IF
		END_IF

		IF bNewMag2 = TRUE THEN
			tyP0203OpsMag2.tyOps.tyBitmapChgMag.usiValueIdx	:= 1;
			IF p_tyDI.bMag2FixedUnclampRS = FALSE OR p_eMagConv2Clp2Status = Error  THEN
				bNewMag2	:= FALSE;
				tyP0203OpsMag2.tyOps.tyBtnChgMag.bValue	:= FALSE;
				tyP0203OpsMag2.tyOps.tyBtnChgMag.bRtLk	:= FALSE;
				tyP0203OpsMag2.tyOps.tyBitmapChgMag.usiValueIdx	:= 0;
			END_IF

		ELSIF bRlsMag2 = TRUE OR bEjectMag2 THEN
			tyP0203OpsMag2.tyOps.tyBitmapChgMag.usiValueIdx	:= 1;
			IF p_tyNtParamCurr.eCustomerReq = Siemens OR p_tyNtParamCurr.eCustomerReq = We_Fabricate THEN
				IF p_bOpsMagConvLD2RlsMagUmask THEN // siemens , read -1 or write TO
					IF p_tyNtParamCurr.eCustomerReq = We_Fabricate THEN
						//bRlsMag2	:= FALSE;
						tyP0203OpsMag2.tyOps.tyBitmapChgMag.usiValueIdx	:= 0;
					END_IF
					tyP0203OpsMag2.tyOps.tyBtnChgMag.bValue	:= FALSE;
					tyP0203OpsMag2.tyOps.tyBtnChgMag.bRtLk	:= FALSE;
				ELSIF p_bOpsMagConvLD2ExtMes THEN //2nd press to eject mag
					bEjectMag2	:= FALSE;
					bRlsMag2	:= FALSE;
					tyP0203OpsMag2.tyOps.tyBtnChgMag.bValue	:= FALSE;
					tyP0203OpsMag2.tyOps.tyBtnChgMag.bRtLk	:= FALSE;
					tyP0203OpsMag2.tyOps.tyBitmapChgMag.usiValueIdx	:= 0;
				ELSIF (p_tyDI.bMag2FixedUnclampRS = TRUE AND p_tyDI.bMagPresentSen2 = FALSE) AND p_tyMcParamCurr.eDSCommA = 0 THEN//smema
					bRlsMag2	:= FALSE;
					tyP0203OpsMag2.tyOps.tyBtnChgMag.bValue	:= FALSE;
					tyP0203OpsMag2.tyOps.tyBtnChgMag.bRtLk	:= FALSE;
					tyP0203OpsMag2.tyOps.tyBitmapChgMag.usiValueIdx	:= 0;
				END_IF

			ELSIF (p_tyDI.bMag2FixedUnclampRS = TRUE AND p_tyDI.bMagPresentSen2 = FALSE) THEN
				bRlsMag2	:= FALSE;
				tyP0203OpsMag2.tyOps.tyBtnChgMag.bValue	:= FALSE;
				tyP0203OpsMag2.tyOps.tyBtnChgMag.bRtLk	:= FALSE;
				tyP0203OpsMag2.tyOps.tyBitmapChgMag.usiValueIdx	:= 0;
			END_IF

		END_IF

		IF p_tyDI.bMagPresentSen2 AND p_tyDI.bMagConvEntSen2 = FALSE THEN
			tyP0203OpsMag2.tyOps.tyBtnChgMag.usiTxtIdx	:= 1;
		ELSE
			tyP0203OpsMag2.tyOps.tyBtnChgMag.usiTxtIdx	:= 0;
			tyP0203OpsMag2.tyOps.tyBtnChgMag.uiMaskRtStat := TRUE;
			IF EDGEPOS(tyP0203OpsMag2.tyOps.tyBtnChgMag.usiTxtIdx =0) THEN
				tyP0203OpsMag2.tyOps.tyBitmapChgMag.usiValueIdx	:= 0;
			END_IF
		END_IF

	//	tyP0203OpsMag2.tyOps.tyBtnChgMag.uiMaskRtStat.0	:= p_bOpsMagConvLD2NewMagAllw OR p_bOpsMagConvLD2RlsMagAllw OR p_bOpsMagConvLD2RlsMagUmask;// OR p_tyDI.bInShutterCloseRS;
		tyP0003MMenu.tyMMenuBtn.tyBtnRlsNewMag2.usiTxtIdx := tyP0003MMenu.tyMMenuBtn.tyBtnRlsNewMagBk2.usiTxtIdx + tyP0203OpsMag2.tyOps.tyBtnChgMag.usiTxtIdx;
		tyP0003MMenu.tyMMenuBtn.tyBtnRlsNewMag2.usiTxtIdx := tyP0003MMenu.tyMMenuBtn.tyBtnRlsNewMagBk2.usiTxtIdx + tyP0203OpsMag2.tyOps.tyBtnChgMag.usiTxtIdx;
		tyP0003MMenu.tyMMenuBtn.tyBtnRlsNewMag2.usiBitmapIdx := tyP0003MMenu.tyMMenuBtn.tyBtnRlsNewMagBk2.usiBitmapIdx + 	tyP0203OpsMag2.tyOps.tyBitmapChgMag.usiValueIdx;
		tyP0003MMenu.tyMMenuBtn.tyBtnRlsNewMag2.uiMaskRtStat := tyP0203OpsMag2.tyOps.tyBtnChgMag.uiMaskRtStat ;
	END_IF
END_ACTION
```

#### Act_EntP0204Disp.st
```iecst
ACTION Act_EntP0204Disp:

	//Access Address
	p_tyC0004Navi ACCESS ADR(tyP0204OpsMag3.tyNaviBack);

	p_tyC0005Main ACCESS ADR(tyCommon.tyMain);

	p_tyC0007Notif ACCESS ADR(tyCommon.tyNotif);

	p_tyC0008MsgBox ACCESS ADR(tyP0204OpsMag3.tyMsgBoxHide);

	p_tyC0009Info ACCESS ADR(tyCommon.tyInfo);

	p_tyC0011RcpPopUp ACCESS ADR(tyP0204OpsMag3.tyRcpPopUp);

	p_tyP0204Ops ACCESS ADR(tyP0204OpsMag3.tyOps);
	p_tyP0204IOMonitor ACCESS ADR(tyP0204OpsMag3.tyIOMonitor);
	p_tyP0204BypsInitConv ACCESS ADR(tyP0204OpsMag3.tyBypsInitConv);
	p_tyP0204Param ACCESS ADR(tyP0204OpsMag3.tyParam);

	//Display
	fUIInRtStatHide(ADR(tyP0204OpsMag3.tyIOMonitor.tyLyr.uiRtStat));
	fUIInRtStatHide(ADR(tyP0204OpsMag3.tyParam.tyLyr.uiRtStat));

	tyP0204OpsMag3.tyOps.tyBtnChgParam.uiRtStat.0	:= NOT(p_tyMcParamCurr.bChgParamEn);
	tyP0204OpsMag3.tyParam.tyNumMaxSlt.diValueMax	:= p_tyMagRcpCurrRcp.diTtlSlt;

	IF p_tyNtParamCurr.bMagAutoVerifyPrep = FALSE THEN
		tyP0204OpsMag3.tyIOMonitor.tyBtnMag3FixedClmpRS.usiTxtIdx	:= 75;
		tyP0204OpsMag3.tyIOMonitor.tyBtnMag3FixedUnclmpRS.usiTxtIdx:= 75;
		tyP0204OpsMag3.tyIOMonitor.tyBtnMag3RmtClmpRS.usiTxtIdx	:= 0;
		tyP0204OpsMag3.tyIOMonitor.tyBtnMag3RmtUnclmpRS.usiTxtIdx:= 0;
		tyP0204OpsMag3.tyIOMonitor.tyBtnMag3FixedClampCtrl.usiTxtIdx:= 41;
		tyP0204OpsMag3.tyIOMonitor.tyBtnMag3RemoteClampCtrl.usiTxtIdx:= 18;
	ELSE
		tyP0204OpsMag3.tyIOMonitor.tyBtnMag3FixedClmpRS.usiTxtIdx	:= 74;
		tyP0204OpsMag3.tyIOMonitor.tyBtnMag3FixedUnclmpRS.usiTxtIdx:= 74;
		tyP0204OpsMag3.tyIOMonitor.tyBtnMag3RmtClmpRS.usiTxtIdx	:= 74;
		tyP0204OpsMag3.tyIOMonitor.tyBtnMag3RmtUnclmpRS.usiTxtIdx:= 74;
		tyP0204OpsMag3.tyIOMonitor.tyBtnMag3FixedClampCtrl.usiTxtIdx:= 41;
		tyP0204OpsMag3.tyIOMonitor.tyBtnMag3RemoteClampCtrl.usiTxtIdx:= 18;

	END_IF

	fUIInRtStatHide(ADR(tyP0204OpsMag3.tyOps.tyBtnAIVWifi.uiRtStat));
	fUIInRtStatHide(ADR(tyP0204OpsMag3.tyOps.tyTxtLblAIV.uiRtStat));

	tyP0204OpsMag3.tyParam.tyNumMaxSlt.diValueMax	:= p_tyMagRcpCurrRcp.diTtlSlt;

END_ACTION
```

#### Act_OptP0204_P0003AIVDat.st
```iecst
ACTION Act_OptP0204_P0003AIVDat:

	//Show Change Mag Button only in Manual Exchane Mode
	tyP0204OpsMag3.tyOps.tyBtnChgMag.uiRtStat.0 := p_tyMcParamCurr.eMagExMode = McSetMagXcAutoMode AND p_tyMcParamCurr.eAGVComProtocol <> McSetAGVCommDisabled OR p_tyNtParamCurr.bProjLifterMagPlatform;;
	tyP0204OpsMag3.tyOps.tyBitmapChgMag.uiRtStat.0 := p_tyMcParamCurr.eMagExMode = McSetMagXcAutoMode AND p_tyMcParamCurr.eAGVComProtocol <> McSetAGVCommDisabled OR p_tyNtParamCurr.bProjLifterMagPlatform;;
	//LED Wifi
	tyP0204OpsMag3.tyOps.tyBtnAIVWifi.bValue	:= p_bAGVOnline;

	//Change Magazine
	IF p_tyNtParamCurr.bProjBtnInsertRmvMag = TRUE THEN

		IF EDGENEG(p_bOpsStatusRun) THEN
			bNewMag3	:= FALSE;
			tyP0204OpsMag3.tyOps.tyBtnChgMag.bRtLk	:= FALSE;
			tyP0204OpsMag3.tyOps.tyBtnChgMag.bRtCompl	:= FALSE;
			tyP0204OpsMag3.tyOps.tyBtnChgMag.bValue		:= FALSE;
		END_IF

		IF tyP0204OpsMag3.tyOps.tyBtnChgMag.bRtCompl = TRUE THEN
			tyP0204OpsMag3.tyOps.tyBitmapChgMag.usiValueIdx	:= 1;
			tyP0204OpsMag3.tyOps.tyBtnChgMag.bRtLk	:= TRUE;
			IF 	p_bOpsMagConvLD3NewMagAllw OR p_bOpsMagConvLD3RlsMagAllw OR p_bOpsMagConvLD3RlsMagUmask THEN
				tyP0204OpsMag3.tyOps.tyBtnChgMag.bRtCompl	:= FALSE;
				bNewMag3	:= p_bOpsMagConvLD3NewMagAllw;
				bRlsMag3	:= p_bOpsMagConvLD3RlsMagAllw;
				bEjectMag3  := p_bOpsMagConvLD3ExtMes;
			END_IF
		END_IF

		IF bNewMag3 = TRUE THEN
			tyP0204OpsMag3.tyOps.tyBitmapChgMag.usiValueIdx	:= 1;
			IF p_tyDI.bMag3FixedUnclampRS = FALSE  OR p_eMagConv2Clp3Status = Error
				THEN
				bNewMag3	:= FALSE;
				tyP0204OpsMag3.tyOps.tyBtnChgMag.bValue	:= FALSE;
				tyP0204OpsMag3.tyOps.tyBtnChgMag.bRtLk	:= FALSE;
				tyP0204OpsMag3.tyOps.tyBitmapChgMag.usiValueIdx	:= 0;
			END_IF

		ELSIF bRlsMag3 = TRUE OR bEjectMag3 THEN
			tyP0204OpsMag3.tyOps.tyBitmapChgMag.usiValueIdx	:= 1;
			IF p_tyNtParamCurr.eCustomerReq = Siemens OR p_tyNtParamCurr.eCustomerReq = We_Fabricate THEN
				IF p_bOpsMagConvLD3RlsMagUmask THEN // siemens , read -1 or write TO
					IF p_tyNtParamCurr.eCustomerReq = We_Fabricate THEN
						//bRlsMag3	:= FALSE;
						tyP0204OpsMag3.tyOps.tyBitmapChgMag.usiValueIdx	:= 0;
						END_IF
					tyP0204OpsMag3.tyOps.tyBtnChgMag.bValue	:= FALSE;
					tyP0204OpsMag3.tyOps.tyBtnChgMag.bRtLk	:= FALSE;
				ELSIF p_bOpsMagConvLD3ExtMes THEN //2nd press to eject mag
					bEjectMag3	:= FALSE;
					bRlsMag3	:= FALSE;
					tyP0204OpsMag3.tyOps.tyBtnChgMag.bValue	:= FALSE;
					tyP0204OpsMag3.tyOps.tyBtnChgMag.bRtLk	:= FALSE;
					tyP0204OpsMag3.tyOps.tyBitmapChgMag.usiValueIdx	:= 0;
				ELSIF(p_tyDI.bMag3FixedUnclampRS = TRUE AND p_tyDI.bMagPresentSen3 = FALSE) AND p_tyMcParamCurr.eDSCommA = 0 THEN//smema
					bRlsMag3	:= FALSE;
					tyP0204OpsMag3.tyOps.tyBtnChgMag.bValue	:= FALSE;
					tyP0204OpsMag3.tyOps.tyBtnChgMag.bRtLk	:= FALSE;
					tyP0204OpsMag3.tyOps.tyBitmapChgMag.usiValueIdx	:= 0;
				END_IF

			ELSIF(p_tyDI.bMag3FixedUnclampRS = TRUE AND p_tyDI.bMagPresentSen3 = FALSE) THEN
				bRlsMag3	:= FALSE;
				tyP0204OpsMag3.tyOps.tyBtnChgMag.bValue	:= FALSE;
				tyP0204OpsMag3.tyOps.tyBtnChgMag.bRtLk	:= FALSE;
				tyP0204OpsMag3.tyOps.tyBitmapChgMag.usiValueIdx	:= 0;
			END_IF

		END_IF

		IF p_tyDI.bMagPresentSen3 AND p_tyDI.bMagConvEntSen3 = FALSE THEN
			tyP0204OpsMag3.tyOps.tyBtnChgMag.usiTxtIdx	:= 1;

		ELSE
			tyP0204OpsMag3.tyOps.tyBtnChgMag.usiTxtIdx	:= 0;

			tyP0204OpsMag3.tyOps.tyBtnChgMag.uiMaskRtStat := TRUE;
			IF EDGEPOS(tyP0204OpsMag3.tyOps.tyBtnChgMag.usiTxtIdx =0) THEN
				tyP0204OpsMag3.tyOps.tyBitmapChgMag.usiValueIdx	:= 0;
		END_IF	END_IF

	//	tyP0204OpsMag3.tyOps.tyBtnChgMag.uiMaskRtStat.0	:= p_bOpsMagConvLD3NewMagAllw OR p_bOpsMagConvLD3RlsMagAllw OR p_bOpsMagConvLD3RlsMagUmask;// OR p_tyDI.bInShutterCloseRS;

		//update for P0003
		tyP0003MMenu.tyMMenuBtn.tyBtnRlsNewMag3.usiTxtIdx := tyP0003MMenu.tyMMenuBtn.tyBtnRlsNewMagBk3.usiTxtIdx + tyP0204OpsMag3.tyOps.tyBtnChgMag.usiTxtIdx;
		tyP0003MMenu.tyMMenuBtn.tyBtnRlsNewMag3.usiTxtIdx := tyP0003MMenu.tyMMenuBtn.tyBtnRlsNewMagBk3.usiTxtIdx + tyP0204OpsMag3.tyOps.tyBtnChgMag.usiTxtIdx;
		tyP0003MMenu.tyMMenuBtn.tyBtnRlsNewMag3.usiBitmapIdx := tyP0003MMenu.tyMMenuBtn.tyBtnRlsNewMagBk3.usiBitmapIdx + 	tyP0204OpsMag3.tyOps.tyBitmapChgMag.usiValueIdx;
		tyP0003MMenu.tyMMenuBtn.tyBtnRlsNewMag3.uiMaskRtStat := tyP0204OpsMag3.tyOps.tyBtnChgMag.uiMaskRtStat ;

	END_IF

END_ACTION
```

#### Act_OptP0204AIVDat.st
```iecst
ACTION Act_OptP0204AIVDat:

	//Show Change Mag Button only in Manual Exchane Mode
	tyP0204OpsMag3.tyOps.tyBtnChgMag.uiRtStat.0 := p_tyMcParamCurr.eMagExMode = McSetMagXcAutoMode AND p_tyMcParamCurr.eAGVComProtocol <> McSetAGVCommDisabled OR p_tyNtParamCurr.bProjLifterMagPlatform;;
	tyP0204OpsMag3.tyOps.tyBitmapChgMag.uiRtStat.0 := p_tyMcParamCurr.eMagExMode = McSetMagXcAutoMode AND p_tyMcParamCurr.eAGVComProtocol <> McSetAGVCommDisabled OR p_tyNtParamCurr.bProjLifterMagPlatform;;
	//LED Wifi
	tyP0204OpsMag3.tyOps.tyBtnAIVWifi.bValue	:= p_bAGVOnline;

	//Change Magazine
	IF p_tyNtParamCurr.bProjBtnInsertRmvMag = TRUE THEN

		IF EDGENEG(p_bOpsStatusRun) THEN
			bNewMag3	:= FALSE;
			tyP0204OpsMag3.tyOps.tyBtnChgMag.bRtLk	:= FALSE;
			tyP0204OpsMag3.tyOps.tyBtnChgMag.bRtCompl	:= FALSE;
			tyP0204OpsMag3.tyOps.tyBtnChgMag.bValue		:= FALSE;
		END_IF

		IF tyP0204OpsMag3.tyOps.tyBtnChgMag.bRtCompl = TRUE THEN
			tyP0204OpsMag3.tyOps.tyBitmapChgMag.usiValueIdx	:= 1;
			tyP0204OpsMag3.tyOps.tyBtnChgMag.bRtLk	:= TRUE;
			IF 	p_bOpsMagConvLD3NewMagAllw OR p_bOpsMagConvLD3RlsMagAllw OR p_bOpsMagConvLD3RlsMagUmask THEN
				tyP0204OpsMag3.tyOps.tyBtnChgMag.bRtCompl	:= FALSE;
				bNewMag3	:= p_bOpsMagConvLD3NewMagAllw;
				bRlsMag3	:= p_bOpsMagConvLD3RlsMagAllw;
				bEjectMag3  := p_bOpsMagConvLD3ExtMes;
			END_IF
		END_IF

		IF bNewMag3 = TRUE THEN
			tyP0204OpsMag3.tyOps.tyBitmapChgMag.usiValueIdx	:= 1;
			IF p_tyDI.bMag3FixedUnclampRS = FALSE  OR p_eMagConv2Clp3Status = Error
				THEN
				bNewMag3	:= FALSE;
				tyP0204OpsMag3.tyOps.tyBtnChgMag.bValue	:= FALSE;
				tyP0204OpsMag3.tyOps.tyBtnChgMag.bRtLk	:= FALSE;
				tyP0204OpsMag3.tyOps.tyBitmapChgMag.usiValueIdx	:= 0;
			END_IF

		ELSIF bRlsMag3 = TRUE OR bEjectMag3 THEN
			tyP0204OpsMag3.tyOps.tyBitmapChgMag.usiValueIdx	:= 1;
			IF p_tyNtParamCurr.eCustomerReq = Siemens OR p_tyNtParamCurr.eCustomerReq = We_Fabricate THEN
				IF p_bOpsMagConvLD3RlsMagUmask THEN // siemens , read -1 or write TO
					IF p_tyNtParamCurr.eCustomerReq = We_Fabricate THEN
						//bRlsMag3	:= FALSE;
						tyP0204OpsMag3.tyOps.tyBitmapChgMag.usiValueIdx	:= 0;
						END_IF
					tyP0204OpsMag3.tyOps.tyBtnChgMag.bValue	:= FALSE;
					tyP0204OpsMag3.tyOps.tyBtnChgMag.bRtLk	:= FALSE;
				ELSIF p_bOpsMagConvLD3ExtMes THEN //2nd press to eject mag
					bEjectMag3	:= FALSE;
					bRlsMag3	:= FALSE;
					tyP0204OpsMag3.tyOps.tyBtnChgMag.bValue	:= FALSE;
					tyP0204OpsMag3.tyOps.tyBtnChgMag.bRtLk	:= FALSE;
					tyP0204OpsMag3.tyOps.tyBitmapChgMag.usiValueIdx	:= 0;
				ELSIF(p_tyDI.bMag3FixedUnclampRS = TRUE AND p_tyDI.bMagPresentSen3 = FALSE) AND p_tyMcParamCurr.eDSCommA = 0 THEN//smema
					bRlsMag3	:= FALSE;
					tyP0204OpsMag3.tyOps.tyBtnChgMag.bValue	:= FALSE;
					tyP0204OpsMag3.tyOps.tyBtnChgMag.bRtLk	:= FALSE;
					tyP0204OpsMag3.tyOps.tyBitmapChgMag.usiValueIdx	:= 0;
				END_IF

			ELSIF(p_tyDI.bMag3FixedUnclampRS = TRUE AND p_tyDI.bMagPresentSen3 = FALSE) THEN
				bRlsMag3	:= FALSE;
				tyP0204OpsMag3.tyOps.tyBtnChgMag.bValue	:= FALSE;
				tyP0204OpsMag3.tyOps.tyBtnChgMag.bRtLk	:= FALSE;
				tyP0204OpsMag3.tyOps.tyBitmapChgMag.usiValueIdx	:= 0;
			END_IF

		END_IF

		IF p_tyDI.bMagPresentSen3 AND p_tyDI.bMagConvEntSen3 = FALSE THEN
			tyP0204OpsMag3.tyOps.tyBtnChgMag.usiTxtIdx	:= 1;
		ELSE
			tyP0204OpsMag3.tyOps.tyBtnChgMag.usiTxtIdx	:= 0;
			tyP0204OpsMag3.tyOps.tyBtnChgMag.uiMaskRtStat := TRUE;
			IF EDGEPOS(tyP0204OpsMag3.tyOps.tyBtnChgMag.usiTxtIdx =0) THEN
				tyP0204OpsMag3.tyOps.tyBitmapChgMag.usiValueIdx	:= 0;
		END_IF	END_IF

	//	tyP0204OpsMag3.tyOps.tyBtnChgMag.uiMaskRtStat.0	:= p_bOpsMagConvLD3NewMagAllw OR p_bOpsMagConvLD3RlsMagAllw OR p_bOpsMagConvLD3RlsMagUmask;// OR p_tyDI.bInShutterCloseRS;

	END_IF
END_ACTION
```

#### Act_OptP0204ChgParam.st
```iecst
ACTION Act_OptP0204ChgParam:

	tyP0204OpsMag3.tyParam.tyNumMinSlt.diValueMax		:= tyP0204OpsMag3.tyParam.tyNumMaxSlt.diValue;
	tyP0204OpsMag3.tyParam.tyNumMaxSlt.diValueMin		:= tyP0204OpsMag3.tyParam.tyNumMinSlt.diValue;
	tyP0204OpsMag3.tyParam.tyNumPitch.diValueMax		:= tyP0204OpsMag3.tyParam.tyNumMaxSlt.diValue - tyP0204OpsMag3.tyParam.tyNumMinSlt.diValue + 1;
	tyP0204OpsMag3.tyParam.tyNumPitch.diValueMin		:= 1;

	tyP0204OpsMag3.tyParam.tyNumMinSltRear.diValueMax		:= tyP0204OpsMag3.tyParam.tyNumMaxSltRear.diValue;
	tyP0204OpsMag3.tyParam.tyNumMaxSltRear.diValueMin		:= tyP0204OpsMag3.tyParam.tyNumMinSltRear.diValue;
	tyP0204OpsMag3.tyParam.tyNumPitchRear.diValueMax		:= tyP0204OpsMag3.tyParam.tyNumMaxSltRear.diValue - tyP0204OpsMag3.tyParam.tyNumMinSltRear.diValue + 1;
	tyP0204OpsMag3.tyParam.tyNumPitchRear.diValueMin		:= 1;

	tyP0204OpsMag3.tyParam.tyNumMtrPshrExtSpd.diValueMin	:= p_tyNtParamCurr.tyProdRcpMtrPshrExtSpd.diMin;
	tyP0204OpsMag3.tyParam.tyNumMtrPshrExtSpd.diValueMax	:= p_tyNtParamCurr.tyProdRcpMtrPshrExtSpd.diMax;
	tyP0204OpsMag3.tyParam.tyNumMtrPshrExtTorq.diValueMin	:= p_tyNtParamCurr.tyProdRcpMtrPshrExtTorq.diMin;
	tyP0204OpsMag3.tyParam.tyNumMtrPshrExtTorq.diValueMax	:= p_tyNtParamCurr.tyProdRcpMtrPshrExtTorq.diMax;
	tyP0204OpsMag3.tyParam.tyNumPshrOffset.diValueMin		:= -(p_tyProdRcpCurrRcp2.diWidthInUM/2-p_tyMcParamCurr.diAWPusherAtHmPosInUM-5000 );
	tyP0204OpsMag3.tyParam.tyNumPshrOffset.diValueMax		:= (p_tyProdRcpCurrRcp2.diWidthInUM/2-p_tyMcParamCurr.diAWPusherAtHmPosInUM-5000 );

	//Control
	IF tyP0204OpsMag3.tyOps.tyBtnChgParam.bRtCompl = TRUE THEN
		tyP0204OpsMag3.tyOps.tyBtnChgParam.bRtCompl	:= FALSE;

		tyProdRcpCurrRcpWr	:= p_tyProdRcpCurrRcp0;

		tyP0204OpsMag3.tyParam.tyDrpDnMcMode.usiValueIdx	:= p_tyProdRcpCurrRcp0.usiMcMod;
		tyP0204OpsMag3.tyParam.tyNumMinSlt.diValue	:= p_tyProdRcpCurrRcp0.diMinSltValue;
		tyP0204OpsMag3.tyParam.tyNumMaxSlt.diValue	:= p_tyProdRcpCurrRcp0.diMaxSltValue;
		tyP0204OpsMag3.tyParam.tyNumPitch.diValue		:= p_tyProdRcpCurrRcp0.diPitch;

		tyP0204OpsMag3.tyParam.tyNumMinSltRear.diValue	:= p_tyProdRcpCurrRcp0.diMinSltValueRear;
		tyP0204OpsMag3.tyParam.tyNumMaxSltRear.diValue	:= p_tyProdRcpCurrRcp0.diMaxSltValueRear;
		tyP0204OpsMag3.tyParam.tyNumPitchRear.diValue		:= p_tyProdRcpCurrRcp0.diPitchRear;

		tyP0204OpsMag3.tyParam.tyNumMtrPshrExtSpd.diValue		:= p_tyProdRcpCurrRcp0.diMtrPshrExtSpd;
		tyP0204OpsMag3.tyParam.tyNumMtrPshrExtTorq.diValue	:= p_tyProdRcpCurrRcp0.diMtrPshrExtTorq;
		tyP0204OpsMag3.tyParam.tyNumPshrOffset.diValue		:= p_tyProdRcpCurrRcp0.diPshrOffset;

		fUIInRtStatOff(ADR(tyP0204OpsMag3.tyParam.tyLyr.uiRtStat));

	END_IF

	tyP0204OpsMag3.tyOps.tyBtnChgParam.bValue	:= tyP0204OpsMag3.tyParam.tyLyr.uiRtStat.0 = FALSE;

	IF tyP0204OpsMag3.tyParam.tyLyr.uiRtStat.0 = FALSE THEN

		IF tyP0204OpsMag3.tyParam.tyBtnSave.bRtCompl = TRUE THEN

			tyProdRcpCurrRcpWr.usiMcMod	:= tyP0204OpsMag3.tyParam.tyDrpDnMcMode.usiValueIdx;
			tyProdRcpCurrRcpWr.diMinSltValue := tyP0204OpsMag3.tyParam.tyNumMinSlt.diValue;
			tyProdRcpCurrRcpWr.diMaxSltValue := tyP0204OpsMag3.tyParam.tyNumMaxSlt.diValue;
			tyProdRcpCurrRcpWr.diPitch := tyP0204OpsMag3.tyParam.tyNumPitch.diValue;

			tyProdRcpCurrRcpWr.diMinSltValueRear := tyP0204OpsMag3.tyParam.tyNumMinSltRear.diValue;
			tyProdRcpCurrRcpWr.diMaxSltValueRear := tyP0204OpsMag3.tyParam.tyNumMaxSltRear.diValue;
			tyProdRcpCurrRcpWr.diPitchRear := tyP0204OpsMag3.tyParam.tyNumPitchRear.diValue;

			tyProdRcpCurrRcpWr.diMtrPshrExtSpd := tyP0204OpsMag3.tyParam.tyNumMtrPshrExtSpd.diValue;
			tyProdRcpCurrRcpWr.diMtrPshrExtTorq := tyP0204OpsMag3.tyParam.tyNumMtrPshrExtTorq.diValue;
			tyProdRcpCurrRcpWr.diPshrOffset := tyP0204OpsMag3.tyParam.tyNumPshrOffset.diValue;

			eProdRcpAct	:= ProdRcpActWriteCurrRcpParam;

			IF p_eProdRcpStatus = Done AND p_eProdRcpStat = ProdRcpActWriteCurrRcpParam THEN
				eProdRcpAct	:= ProdRcpActIdle;

				//UIP0400
				tyP0400ProdSel.tyProdSel.tyTxtMcMode.usiValueIdx	:= p_tyProdRcpCurrRcp0.usiMcMod;

				tyP0400ProdSel.tyProdSel.tyNumMinSlt.diValue	:= p_tyProdRcpCurrRcp0.diMinSltValue;
				tyP0400ProdSel.tyProdSel.tyNumMaxSlt.diValue	:= p_tyProdRcpCurrRcp0.diMaxSltValue;
				tyP0400ProdSel.tyProdSel.tyNumPitch.diValue		:= p_tyProdRcpCurrRcp0.diPitch;

				tyP0400ProdSel.tyProdSel.tyNumMinSltRear.diValue	:= p_tyProdRcpCurrRcp0.diMinSltValueRear;
				tyP0400ProdSel.tyProdSel.tyNumMaxSltRear.diValue	:= p_tyProdRcpCurrRcp0.diMaxSltValueRear;
				tyP0400ProdSel.tyProdSel.tyNumPitchRear.diValue		:= p_tyProdRcpCurrRcp0.diPitchRear;

				tyP0400ProdSel.tyProdSel.tyNumMtrPshrExtSpd.diValue		:= p_tyProdRcpCurrRcp0.diMtrPshrExtSpd;
				tyP0400ProdSel.tyProdSel.tyNumMtrPshrExtTorq.diValue	:= p_tyProdRcpCurrRcp0.diMtrPshrExtTorq;
				tyP0400ProdSel.tyProdSel.tyNumPshrOffset.diValue		:= p_tyProdRcpCurrRcp0.diPshrOffset;

				tyP0204OpsMag3.tyParam.tyBtnSave.bRtCompl	:= FALSE;
				tyP0204OpsMag3.tyParam.tyBtnSave.bValue		:= FALSE;

				fUIInRtStatHide(ADR(tyP0204OpsMag3.tyParam.tyLyr.uiRtStat));

			ELSIF p_eProdRcpStatus = Error THEN
				p_tyC0008MsgBox ACCESS ADR(tyP0204OpsMag3.tyMsgBoxSaveErr);

				IF tyP0204OpsMag3.tyMsgBoxSaveErr.tyBtnNo.bRtCompl = TRUE THEN
					tyP0204OpsMag3.tyMsgBoxSaveErr.tyBtnNo.bRtCompl	:= FALSE;
					tyP0204OpsMag3.tyMsgBoxSaveErr.tyBtnNo.bValue	:= FALSE;

					p_tyC0008MsgBox ACCESS ADR(tyP0204OpsMag3.tyMsgBoxHide);

					//Restore Param
					tyProdRcpCurrRcpWr	:= p_tyProdRcpCurrRcp2;

					tyP0204OpsMag3.tyParam.tyBtnSave.bRtCompl		:= FALSE;
					tyP0204OpsMag3.tyParam.tyBtnSave.bValue			:= FALSE;

					fUIInRtStatHide(ADR(tyP0204OpsMag3.tyParam.tyLyr.uiRtStat));

				END_IF

			END_IF

		ELSIF tyP0204OpsMag3.tyParam.tyBtnCancel.bRtCompl = TRUE THEN
			tyP0204OpsMag3.tyParam.tyBtnCancel.bRtCompl				:= FALSE;
			tyP0204OpsMag3.tyParam.tyBtnCancel.bValue				:= FALSE;

			fUIInRtStatHide(ADR(tyP0204OpsMag3.tyParam.tyLyr.uiRtStat));

		END_IF

	END_IF

	//Mask
	tyP0204OpsMag3.tyOps.tyBtnChgParam.uiMaskRtStat.0	:= p_tyUsrMgmtCurrAccessRgt.bChgParam AND p_bOpsStatusStop;

END_ACTION
```

#### Act_OptP0204InsertRmvMag.st
```iecst
ACTION Act_OptP0204InsertRmvMag:

	//Insert & Removed Magazine Manually Without Button Control
//	IF p_tyNtParamCurr.bProjBtnInsertRmvMag = FALSE THEN
//
//		IF p_bOpsStatusRun AND p_bOpsMagConvLD3InitDone THEN
//
//			fbMag3EntrySenOnTm(IN := p_tyDI.bMagPresentSen3 OR p_tyDI.bMagConvEntSen3);
//
//			IF bNewMag3 = FALSE AND bRlsMag3 = FALSE THEN
//				IF p_bOpsMagConvLD3NewMagAllw AND fbMag3EntrySenOnTm.Q AND NOT p_bOpsMagConvLD3MagExitedWait THEN
//					bNewMag3	:= TRUE;
//				END_IF
//
//				IF p_bOpsMagConvLD3RlsMagAllw AND p_tyDI.bMagPresentSen3 AND p_tyDI.bInShutterCloseRS AND p_tyBuffer3BffrStat.bBffrMty THEN
//					bRlsMag3	:= TRUE;
//				END_IF
//			END_IF
//
//			IF bNewMag3 = TRUE THEN
//
//				IF p_tyDI.bMag3FixedClampRS = TRUE AND p_tyDI.bMag3RemoteClampRS = TRUE THEN
//					bNewMag3	:= FALSE;
//				END_IF
//
//			ELSIF bRlsMag3 = TRUE THEN
//
//				IF p_tyDI.bMag3FixedUnclampRS = TRUE AND p_tyDI.bMag3RemoteUnclampRS = TRUE AND p_tyDI.bMagConvEntSen3 = TRUE THEN
//					bRlsMag3	:= FALSE;
//				END_IF
//
//			END_IF
//
//		ELSE
//
//			bNewMag3	:= FALSE;
//			bRlsMag3	:= FALSE;
//
//			fbMag3EntrySenOnTm(IN := FALSE);
//
//		END_IF
//
//	END_IF

END_ACTION
```

#### Act_OptP0204IOMonitor.st
```iecst
ACTION Act_OptP0204IOMonitor:

	IF tyP0204OpsMag3.tyOps.tyHotspotIOMonitor.bRtCompl = TRUE THEN
		tyP0204OpsMag3.tyOps.tyHotspotIOMonitor.bRtCompl	:= FALSE;

		fUIInRtStatOff(ADR(tyP0204OpsMag3.tyIOMonitor.tyLyr.uiRtStat));

		p_tyC0004Navi ACCESS ADR(tyP0204OpsMag3.tyNaviHide);

	ELSIF tyP0204OpsMag3.tyIOMonitor.tyHotspotClose.bRtCompl = TRUE THEN
		tyP0204OpsMag3.tyIOMonitor.tyHotspotClose.bRtCompl	:= FALSE;

		fUIInRtStatHide(ADR(tyP0204OpsMag3.tyIOMonitor.tyLyr.uiRtStat));

		p_tyC0004Navi ACCESS ADR(tyP0204OpsMag3.tyNaviBack);

	END_IF

	IF tyP0204OpsMag3.tyIOMonitor.tyLyr.uiRtStat.0 = FALSE THEN

		//Digital Input
		tyP0204OpsMag3.tyIOMonitor.tyBtnSafetyRlySig.bValue				:= p_tyDI.bSafetyRlySig;
		tyP0204OpsMag3.tyIOMonitor.tyBtnEStop.bValue					:= p_tyDI.bEStopSig;
		tyP0204OpsMag3.tyIOMonitor.tyBtnCoverSWSig.bValue				:= p_tyDI.bCoverSWSig;
		tyP0204OpsMag3.tyIOMonitor.tyBtnDSBA.bValue						:= p_tyDI.bDSBA;
		tyP0204OpsMag3.tyIOMonitor.tyBtnDSBB.bValue						:= p_tyDI.bDSBB;
		tyP0204OpsMag3.tyIOMonitor.tyBtnMag3FixedClmpRS.bValue			:= p_tyDI.bMag3FixedClampRS;
		tyP0204OpsMag3.tyIOMonitor.tyBtnMag3FixedUnclmpRS.bValue		:= p_tyDI.bMag3FixedUnclampRS;
		tyP0204OpsMag3.tyIOMonitor.tyBtnMag3RmtClmpRS.bValue			:= p_tyDI.bMag3RemoteClampRS;
		tyP0204OpsMag3.tyIOMonitor.tyBtnMag3RmtUnclmpRS.bValue			:= p_tyDI.bMag3RemoteUnclampRS;
		tyP0204OpsMag3.tyIOMonitor.tyBtnMag3ConvEntrySen.bValue			:= p_tyDI.bMagConvEntSen3;
		tyP0204OpsMag3.tyIOMonitor.tyBtnMag3PresentSen.bValue			:= p_tyDI.bMagPresentSen3;
		tyP0204OpsMag3.tyIOMonitor.tyBtnMag3AIVInPosSen1.bValue			:= p_tyDI.bMag3AGVInPosSen1;
		tyP0204OpsMag3.tyIOMonitor.tyBtnMag3AIVInPosSen2.bValue			:= p_tyDI.bMag3AGVInPosSen2;
		tyP0204OpsMag3.tyIOMonitor.tyBtnMag3OrientationChkSen1.bValue	:= p_tyDI.bMag3OrientChkSen1;
		tyP0204OpsMag3.tyIOMonitor.tyBtnMag3OrientationChkSen2.bValue	:= p_tyDI.bMag3OrientChkSen2;

		tyP0204OpsMag3.tyIOMonitor.tyBtnSelUnclampRS.bValue				:= p_tyDI.bMag3SelUnClampRS;

		tyP0204OpsMag3.tyIOMonitor.tyBtnCAB717Sen.bValue				:= p_tyDI.bMagConvCAB717MagSen3;
		tyP0204OpsMag3.tyIOMonitor.tyBtnHeightSen.bValue				:= p_tyDI.bMagConvHeightSen3 OR p_tyDI.bHighMagDetSen3;
		tyP0204OpsMag3.tyIOMonitor.tyBtnMagSmallSen.bValue				:= p_tyDI.bMagConvSmallMagSen3;
		tyP0204OpsMag3.tyIOMonitor.tyBtnMagLargeSen.bValue				:= p_tyDI.bMagConvLargeMagSen3;
		tyP0204OpsMag3.tyIOMonitor.tyBtnMagDetSen.bValue				:= p_tyDI.bMag3FixedSideDetect;

		//Digital Output
		tyP0204OpsMag3.tyIOMonitor.tyBtnSafetyRlyRst.bValue				:= p_tyDO.bSafetyRlyRst;
		tyP0204OpsMag3.tyIOMonitor.tyBtnTLGreen.bValue					:= p_tyDO.bTLGreen;
		tyP0204OpsMag3.tyIOMonitor.tyBtnTLAmber.bValue					:= p_tyDO.bTLAmber;
		tyP0204OpsMag3.tyIOMonitor.tyBtnTLRed.bValue					:= p_tyDO.bTLRed;
		tyP0204OpsMag3.tyIOMonitor.tyBtnBuzzer.bValue					:= p_tyDO.bBuzzer;
		tyP0204OpsMag3.tyIOMonitor.tyBtnDBAA.bValue						:= p_tyDO.bDBAA;
		tyP0204OpsMag3.tyIOMonitor.tyBtnDBAB.bValue						:= p_tyDO.bDBAB;
		tyP0204OpsMag3.tyIOMonitor.tyBtnMag3FixedClampCtrl.bValue		:= p_tyDO.bMag3FixedClampCtrl;
		tyP0204OpsMag3.tyIOMonitor.tyBtnMag3RemoteClampCtrl.bValue		:= p_tyDO.bMag3RemoteClampCtrl;
		tyP0204OpsMag3.tyIOMonitor.tyBtnMag3ConvMtrIn.bValue			:= p_tyDO.bMag3ConvMtrIn;
		tyP0204OpsMag3.tyIOMonitor.tyBtnMag3ConvMtrOut.bValue			:= p_tyDO.bMag3ConvMtrOut;
		tyP0204OpsMag3.tyIOMonitor.tyBtnMagSelClampCtrl.bValue			:= p_tyDO.bMag3SelClampCtrl;
	END_IF

END_ACTION
```

#### Act_OptP0204UpdtDat.st
```iecst
ACTION Act_OptP0204UpdtDat:

	//Status
	fbMcStatUpdtTm(IN := TRUE);
	IF fbMcStatUpdtTm.Q = TRUE THEN
		fbMcStatUpdtTm(IN := FALSE);

		IF p_tyNtParamCurr.bProjLifterMagPlatform THEN
			tyP0204OpsMag3.tyOps.tyStringMcStat.sValue	:= p_sOpsLifMagLDStepTxt;
		ELSE
			tyP0204OpsMag3.tyOps.tyStringMcStat.sValue	:= p_sOpsMagConvLD3StepTxt;
		END_IF

	END_IF

	//Mode
	tyP0204OpsMag3.tyOps.tyTxtMod.usiValueIdx	:= p_tyProdRcpCurrRcp1.usiMcMod;

	//Width
	IF p_tyNtParamCurr.bAWPrep = TRUE AND p_tyMcParamCurr.bAWDis = FALSE THEN
		tyP0204OpsMag3.tyOps.tyNumWidth.diValue	:= p_tyMcParamCurr.diWidthAtHmPosInUM - p_diAWOpenActualPos;
		tyP0204OpsMag3.tyOps.tyNumWidth2.diValue	:= p_tyMcParamCurr.diWidthAtHmPosInUM - p_diAWOpenActualPos;
	ELSE
		tyP0204OpsMag3.tyOps.tyNumWidth.diValue	:= p_tyProdRcpCurrRcp1.diWidthInUM;
		tyP0204OpsMag3.tyOps.tyNumWidth2.diValue	:= p_tyProdRcpCurrRcp1.diWidthInUM2;
	END_IF

	//Program Info
	IF p_tyNtParamCurr.eProjMag <> LDMagQuadruple THEN
		IF p_tyNtParamCurr.bProjAutoRcpPrep AND p_tyMcParamCurr.bHermesSvyEn THEN
			tyP0204OpsMag3.tyOps.tyNumMinSltRange.diValue		:= p_diLinkAutoRcpMag3MinSlt;
			tyP0204OpsMag3.tyOps.tyNumMaxSltRange.diValue		:= p_diLinkAutoRcpMag3MaxSlt;
			tyP0204OpsMag3.tyOps.tyNumPitch.diValue				:= p_diLinkAutoRcpMag3Pitch;
			tyP0204OpsMag3.tyOps.tyStringProdNm.sValue			:= p_tyAutoRcpMagRcp[3].sWorkOrderId;
		ELSE
			tyP0204OpsMag3.tyOps.tyNumMinSltRange.diValue		:= p_tyProdRcpCurrRcp2.diMinSltValue;
			tyP0204OpsMag3.tyOps.tyNumMaxSltRange.diValue		:= p_tyProdRcpCurrRcp2.diMaxSltValue;
			tyP0204OpsMag3.tyOps.tyNumPitch.diValue				:= p_tyProdRcpCurrRcp2.diPitch;
			tyP0204OpsMag3.tyOps.tyStringProdNm.sValue			:= p_tyProdRcpCurrRcp2.sRcpNm;
		END_IF
		tyP0204OpsMag3.tyOps.tyBtnToptoBtm.bValue			:= p_tyProdRcpCurrRcp2.bTopToBtm;
		//Magazine Info
		tyP0204OpsMag3.tyOps.tyStringMagNm.sValue	:= p_tyMagRcpCurrRcp.sRcpNm;
	ELSE
		CASE p_tyProdRcpCurrRcp2.usiMcMod OF
			0:
				tyP0204OpsMag3.tyOps.tyStringProdNm.sValue		:= p_tyProdRcpCurrRcp2.sRcpNm;
				tyP0204OpsMag3.tyOps.tyNumMinSltRange.diValue		:= p_tyProdRcpCurrRcp2.diMinSltValue;
				tyP0204OpsMag3.tyOps.tyNumMaxSltRange.diValue		:= p_tyProdRcpCurrRcp2.diMaxSltValue;
				tyP0204OpsMag3.tyOps.tyBtnToptoBtm.bValue			:= p_tyProdRcpCurrRcp2.bTopToBtm;
				tyP0204OpsMag3.tyOps.tyNumPitch.diValue			:= p_tyProdRcpCurrRcp2.diPitch;
				//Magazine Info
				tyP0204OpsMag3.tyOps.tyStringMagNm.sValue	:= p_tyMagRcpCurrRcp.sRcpNm;

			1,2:

				tyP0204OpsMag3.tyOps.tyStringProdNm.sValue		:= p_tyProdRcpCurrRcp2.sRcpNm;
				tyP0204OpsMag3.tyOps.tyNumMinSltRange.diValue		:= p_tyProdRcpCurrRcp2.diMinSltValueRear;
				tyP0204OpsMag3.tyOps.tyNumMaxSltRange.diValue		:= p_tyProdRcpCurrRcp2.diMaxSltValueRear;
				tyP0204OpsMag3.tyOps.tyBtnToptoBtm.bValue			:= p_tyProdRcpCurrRcp2.bTopToBtm;
				tyP0204OpsMag3.tyOps.tyNumPitch.diValue			:= p_tyProdRcpCurrRcp2.diPitchRear;
				//Magazine Info
				tyP0204OpsMag3.tyOps.tyStringMagNm.sValue	:= p_tyMagRcpCurrRcp1.sRcpNm;
		END_CASE
	END_IF

	//Magazine Info
//	tyP0204OpsMag3.tyOps.tyStringMagNm.sValue	:= p_tyMagRcpCurrRcp.sRcpNm;

	IF p_bBuffer3MagPresent = TRUE THEN
		tyP0204OpsMag3.tyOps.tyNumMag3AvlQty.diValue	:= p_tyBuffer3BffrStat.diTtlGdBrd + p_tyBuffer3BffrStat.diTtlBadBrd;
		tyP0204OpsMag3.tyOps.tyNumMag3TtlSlt.diValue	:= p_tyBuffer3BffrStat.diTtlBrdCap;
	ELSE
		tyP0204OpsMag3.tyOps.tyNumMag3AvlQty.diValue	:= 0;
		tyP0204OpsMag3.tyOps.tyNumMag3TtlSlt.diValue	:= 0;
	END_IF

	//Magazine Present States
	IF p_bBuffer3MagPresent = TRUE THEN

		IF p_tyBuffer3BffrStat.bBffrFull = TRUE THEN
			tyP0204OpsMag3.tyOps.tyTxtMag3Stat.usiValueIdx := 2;
			tyP0204OpsMag3.tyOps.tyTxtMag3Stat.usiColor	   := 0;
		ELSIF p_tyBuffer3BffrStat.bBffrMty = TRUE THEN
			tyP0204OpsMag3.tyOps.tyTxtMag3Stat.usiValueIdx := 1;
			tyP0204OpsMag3.tyOps.tyTxtMag3Stat.usiColor	   := 1;
		ELSE
			tyP0204OpsMag3.tyOps.tyTxtMag3Stat.usiValueIdx := 3;
			tyP0204OpsMag3.tyOps.tyTxtMag3Stat.usiColor	   := 0;
		END_IF

	ELSE
		tyP0204OpsMag3.tyOps.tyTxtMag3Stat.usiValueIdx := 0;
		tyP0204OpsMag3.tyOps.tyTxtMag3Stat.usiColor	   := 1;
	END_IF

	//Product Recipe 254
	tyP0204OpsMag3.tyOps.tyHotspotShowLRcp.uiRtStat.0 := NOT(tyP0204OpsMag3.tyOps.tyStringProdNm.sValue <> '');

	IF tyP0204OpsMag3.tyOps.tyHotspotShowLRcp.bRtCompl = TRUE THEN
		tyP0204OpsMag3.tyOps.tyHotspotShowLRcp.bRtCompl := FALSE;

		fUIInRtStatOff(ADR(tyP0204OpsMag3.tyRcpPopUp.tyLyr.uiRtStat));

		tyP0204OpsMag3.tyRcpPopUp.tyStringInfo.sValue  := p_tyProdRcpCurrRcp1.sRcpNm;

	ELSIF tyP0204OpsMag3.tyRcpPopUp.tyHotspotClose.bRtCompl = TRUE THEN
		tyP0204OpsMag3.tyRcpPopUp.tyHotspotClose.bRtCompl := FALSE;

		fUIInRtStatHide(ADR(tyP0204OpsMag3.tyRcpPopUp.tyLyr.uiRtStat));

	END_IF
END_ACTION
```
